ABB RAPID module: ProgSide1.mod

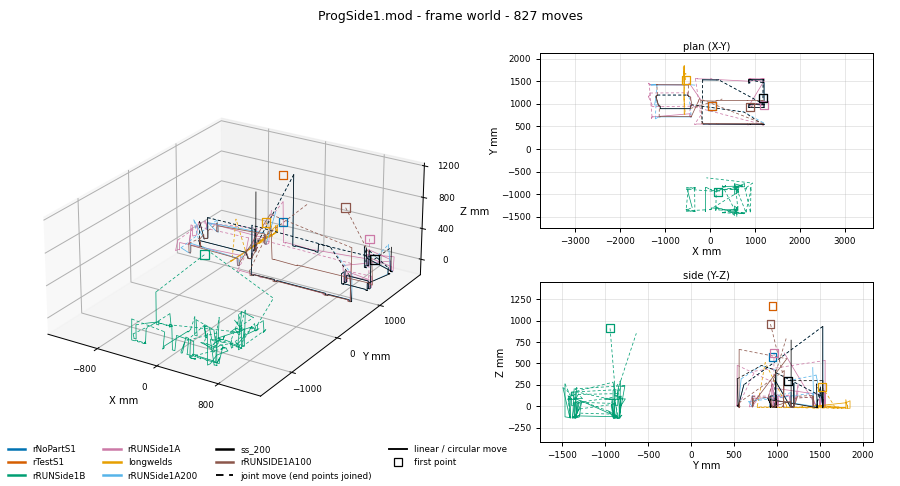
[picture p0: tool path of ProgSide1.mod in frame world, 827 of 843 moves have a stored position in this frame; points joined in program order, loops and branches not executed]
MODULE ProgSide1
    !setup for 300ss
    RECORD WeldPoint300
    robtarget trans;
    robtarget approach;
    robtarget start;
    robtarget end;
    robtarget exitt;
    seamdata seamiii;
    welddata weldiii;
    ENDRECORD
    PERS WeldPoint300 wp300{40};
    PERS num WeldiiiCount := 0;


	!specific zoffset for 200 ss

    TASK PERS wobjdata wobjSide1A200:=[FALSE,TRUE,"",[[0,0,0],[1,0,0,0]],[[0,0,0],[1,0,0,0]]];

    PERS bool bZ_B_onlySide2:=FALSE;
	PERS bool bZ_B_onlySide1:=FALSE;
	PERS bool bC_HalfstepSide2:=FALSE;
	PERS bool bC_HalfstepSide1:=FALSE;
	PERS bool bZ_HalfstepSide1:=FALSE;
	PERS bool bZ_HalfstepSide2:=FALSE;
	PERS bool bAngleSide1:=FALSE;
	PERS bool bAngleSide2:=FALSE;
	PERS bool bTestWeldSide1:=FALSE;
    PERS bool bTestWeldSide2:=FALSE;

    ! Boolian initialization for the SS 300 Frames
    PERS bool bNoPartSide1:=FALSE;
	PERS bool bNoPartSide2:=FALSE;
    PERS bool A_onlySide2:=FALSE;
    PERS bool B_onlySide2:=FALSE;
	PERS bool A_onlySide1:=FALSE;
    PERS bool B_onlySide1:=FALSE;
	PERS bool AB_Side1:=FALSE;
    PERS bool AB_Side2:=FALSE;

    ! Boolian initialization for the SelFrames procedures except the SS 300s.
    PERS bool bSkid50:=FALSE;
    PERS bool bSkid100:=FALSE;
	PERS bool bSkid200:=FALSE;
    PERS bool bSide1A100:=FALSE;
    PERS bool bSide1A200:=FALSE;
    PERS bool bSide1A300:=TRUE;

    PERS bool bRover:=FALSE;
    PERS bool bLongWeld:=FALSE;


	TASK PERS welddata weld7:=[15.24,16.6963,[7,0,0,0,0,0,0,0,0],[7,0,0,0,0,0,0,0,0]];
	TASK PERS welddata weld6:=[16.2983,16.6963,[6,0,0,0,0,0,0,0,0],[6,0,0,0,0,0,0,0,0]];

	CONST robtarget pPounceOS1:=[[-398.58,690.45,580.22],[0.00101632,0.999968,-0.00455572,0.00645523],[-1,0,-1,0],[9E+09,9E+09,9E+09,9E+09,9E+09,9E+09]];
	CONST robtarget pPounceS21:=[[580.19,77.23,83.43],[0.071601,0.767336,-0.436334,0.464416],[-1,0,-2,0],[9E+09,9E+09,9E+09,9E+09,9E+09,9E+09]];
	TASK PERS seamdata seam2:=[4,1,[1,0,52,74.0833,0,0,0,0,0],0,0,0,0,0,[1,0,48,0,0,0,0,0,0],0.01,0.1,[1,0,48,105.833,0,0,0,0,0],0,0,[0,0,0,0,0,0,0,0,0],1];
	TASK PERS seamdata seam10:=[4,1,[1,0,50,80.4333,0,0,0,0,0],0,0,0,0,0,[0,0,0,0,0,0,0,0,0],0.25,0.25,[1,0,50,38.1,0,0,0,0,0],0,0,[0,0,0,0,0,0,0,0,0],1];
	CONST robtarget pPounceS31:=[[358.52,159.10,437.93],[0.0181628,-0.398765,0.916866,0.00362624],[-2,0,-2,0],[9E+09,9E+09,9E+09,9E+09,9E+09,9E+09]];
	CONST robtarget pPounceS41:=[[193.25,136.11,113.74],[0.188325,0.84715,-0.195157,0.45693],[-1,-1,-2,0],[9E+09,9E+09,9E+09,9E+09,9E+09,9E+09]];
	PERS welddata weld11:=[13.5467,0,[1,0,50,84.6667,0,0,0,0,0],[0,0,0,0,0,0,0,0,0]];
	PERS welddata weld10:=[14.8167,0,[1,0,50,95.25,0,0,0,0,0],[0,0,0,0,0,0,0,0,0]];
	TASK PERS seamdata seam11:=[1,1,[1,0,50,84.6667,0,0,0,0,0],0,0,0,0,0,[0,0,0,0,0,0,0,0,0],0,0,[0,0,0,0,0,0,0,0,0],0,0,[0,0,0,0,0,0,0,0,0],0];
	TASK PERS seamdata seam12:=[1,1,[1,0,18.5,381,0,0,0,0,0],0,0,0,0,0,[0,0,0,0,0,0,0,0,0],0,0,[0,0,0,0,0,0,0,0,0],0,0,[0,0,0,0,0,0,0,0,0],0];
	TASK PERS seamdata seam13:=[1,1,[1,0,14,127,0,0,0,0,0],0,0,0,0,0,[0,0,0,0,0,0,0,0,0],0,0,[0,0,0,0,0,0,0,0,0],0,0,[0,0,0,0,0,0,0,0,0],0];
	PERS welddata weld12:=[21.9625,0,[1,0,19,70.6797,0,0,0,0,0],[0,0,0,0,0,0,0,0,0]];
	PERS welddata weld13:=[6.90033,6.90033,[1,0,19,110.71,0,0,0,0,0],[0,0,18.5,110.71,0,0,0,0,0]];
	CONST robtarget pSafeS11:=[[-996.19,963.00,488.78],[0.0459907,-0.688393,0.722625,0.0425673],[1,-1,1,0],[9E+09,9E+09,9E+09,9E+09,9E+09,9E+09]];
	CONST robtarget pSafeS21:=[[-996.19,963.00,488.76],[0.0459983,-0.688397,0.722622,0.0425559],[1,-1,1,0],[9E+09,9E+09,9E+09,9E+09,9E+09,9E+09]];
	CONST robtarget pSafeS31:=[[506.44,675.04,711.34],[0.0314656,-0.935633,0.203865,-0.286426],[0,0,-2,0],[9E+09,9E+09,9E+09,9E+09,9E+09,9E+09]];
	CONST robtarget pSafeS41:=[[488.47,1091.24,654.25],[0.0459806,-0.688392,0.722627,0.0425664],[0,0,-1,0],[9E+09,9E+09,9E+09,9E+09,9E+09,9E+09]];
	CONST robtarget pSafeS51:=[[528.23,1196.89,528.24],[0.224235,-0.753625,-0.525201,-0.325471],[0,-1,-3,0],[9E+09,9E+09,9E+09,9E+09,9E+09,9E+09]];
	CONST robtarget pSafeS61:=[[597.29,1295.03,43.37],[0.191334,-0.732058,-0.538062,-0.371444],[0,-1,-2,0],[9E+09,9E+09,9E+09,9E+09,9E+09,9E+09]];
	CONST robtarget pSafeS71:=[[542.66,1322.39,535.75],[0.223485,-0.764556,-0.487458,-0.357621],[0,-1,-2,0],[9E+09,9E+09,9E+09,9E+09,9E+09,9E+09]];
	CONST robtarget pSafeS81:=[[542.66,1322.38,535.76],[0.223484,-0.764558,-0.487457,-0.35762],[0,-1,-2,0],[9E+09,9E+09,9E+09,9E+09,9E+09,9E+09]];
	CONST robtarget pPounceS51:=[[15.28,993.81,754.75],[0.277209,0.263034,-0.848831,-0.365313],[0,0,0,0],[9E+09,9E+09,9E+09,9E+09,9E+09,9E+09]];
	CONST robtarget pPounceS61:=[[649.55,1131.56,389.19],[0.45355,-0.00505177,-0.879595,-0.143459],[0,0,0,0],[9E+09,9E+09,9E+09,9E+09,9E+09,9E+09]];
	TASK PERS seamdata seam3:=[1,1,[1,0,35,84.6667,0,0,0,0,0],0,0,0,0,0,[1,0,48,0,0,0,0,0,0],0.01,0.1,[1,0,48,105.833,0,0,0,0,0],0,0,[0,0,0,0,0,0,0,0,0],1];
	CONST robtarget pSafeS101:=[[572.94,23.46,738.68],[0.0502756,-0.467207,-0.815726,-0.337314],[0,0,0,0],[9E+09,9E+09,9E+09,9E+09,9E+09,9E+09]];
	CONST robtarget pSafeS111:=[[877.74,-1.14,1156.39],[0.00629855,0.0017594,0.999979,-0.000494623],[0,-1,0,0],[9E+09,9E+09,9E+09,9E+09,9E+09,9E+09]];
	CONST robtarget pSafeS121:=[[877.74,-1.14,1156.39],[0.00629925,0.00175887,0.999979,-0.000492925],[0,-1,0,0],[9E+09,9E+09,9E+09,9E+09,9E+09,9E+09]];
	CONST robtarget pSafeS131:=[[865.02,1139.54,-19.77],[0.144708,-0.274627,0.931028,0.191903],[0,-2,2,0],[9E+09,9E+09,9E+09,9E+09,9E+09,9E+09]];
	CONST robtarget pSafeS141:=[[849.60,1148.97,-24.06],[0.00628216,0.00187497,0.999979,-0.000396021],[0,-1,1,0],[9E+09,9E+09,9E+09,9E+09,9E+09,9E+09]];
	CONST robtarget pSafeS151:=[[1007.97,1505.52,122.27],[0.0460025,-0.688387,0.722632,0.0425454],[0,1,-2,0],[9E+09,9E+09,9E+09,9E+09,9E+09,9E+09]];
	CONST robtarget pHomePos20:=[[365.14,988.92,-33.91],[0.0351389,-0.509982,-0.859022,-0.0276858],[0,-1,1,0],[9E+09,9E+09,9E+09,9E+09,9E+09,9E+09]];
	CONST robtarget pHomePos30:=[[365.15,979.87,-33.91],[0.0351433,-0.509968,-0.85903,-0.0276827],[0,-1,1,0],[9E+09,9E+09,9E+09,9E+09,9E+09,9E+09]];
	CONST robtarget pHomePos40:=[[365.14,979.87,-15.16],[0.0351385,-0.509986,-0.859019,-0.0276867],[0,-1,1,0],[9E+09,9E+09,9E+09,9E+09,9E+09,9E+09]];
	CONST robtarget pHomePos50:=[[433.12,979.73,-15.17],[0.0351369,-0.509964,-0.859032,-0.0276871],[0,-1,1,0],[9E+09,9E+09,9E+09,9E+09,9E+09,9E+09]];
	CONST robtarget pHomePos60:=[[430.57,978.47,-32.25],[0.0351433,-0.50998,-0.859023,-0.0276796],[0,-1,1,0],[9E+09,9E+09,9E+09,9E+09,9E+09,9E+09]];
	CONST robtarget pHomePos70:=[[430.57,978.46,-32.26],[0.0351393,-0.509989,-0.859017,-0.027681],[0,-1,1,0],[9E+09,9E+09,9E+09,9E+09,9E+09,9E+09]];
	CONST robtarget pHomePos80:=[[430.59,974.37,-32.26],[0.0351321,-0.50997,-0.859029,-0.0276862],[0,-1,1,0],[9E+09,9E+09,9E+09,9E+09,9E+09,9E+09]];
	CONST robtarget pHomePos90:=[[430.57,974.36,-24.94],[0.0351397,-0.509992,-0.859016,-0.0276799],[0,-1,1,0],[9E+09,9E+09,9E+09,9E+09,9E+09,9E+09]];
	CONST robtarget pHomePos100:=[[445.83,974.38,-24.94],[0.0351383,-0.509986,-0.859019,-0.0276863],[0,-1,1,0],[9E+09,9E+09,9E+09,9E+09,9E+09,9E+09]];
	CONST robtarget pHomePos110:=[[446.40,974.36,-32.29],[0.0351532,-0.510006,-0.859007,-0.0276708],[0,-1,1,0],[9E+09,9E+09,9E+09,9E+09,9E+09,9E+09]];
	CONST robtarget pHomePos120:=[[446.42,974.37,-32.29],[0.0351424,-0.509994,-0.859014,-0.0276814],[0,-1,1,0],[9E+09,9E+09,9E+09,9E+09,9E+09,9E+09]];
	CONST robtarget pSafeS12:=[[1424.79,-683.57,-13.74],[0.019551,0.168491,0.985501,-0.00412114],[-1,1,-2,0],[9E+09,9E+09,9E+09,9E+09,9E+09,9E+09]];
	CONST robtarget pSafeS22:=[[1462.93,-789.47,-110.40],[0.0637154,0.393325,0.863983,0.307846],[-1,1,-2,0],[9E+09,9E+09,9E+09,9E+09,9E+09,9E+09]];
	CONST robtarget pSafeS32:=[[1462.93,-821.54,-110.39],[0.0637158,0.39332,0.863986,0.307843],[-1,1,-2,0],[9E+09,9E+09,9E+09,9E+09,9E+09,9E+09]];
	CONST robtarget pSafeS42:=[[1462.93,-821.54,-110.39],[0.0637186,0.393326,0.863982,0.307849],[-1,1,-2,0],[9E+09,9E+09,9E+09,9E+09,9E+09,9E+09]];
	CONST robtarget pSafeS52:=[[1462.55,-1477.98,-107.56],[0.0637139,0.393324,0.863983,0.30785],[-1,0,-1,0],[9E+09,9E+09,9E+09,9E+09,9E+09,9E+09]];
	CONST robtarget pSafeS62:=[[1462.54,-1515.56,-107.57],[0.0637098,0.393325,0.863984,0.307846],[-1,0,-1,0],[9E+09,9E+09,9E+09,9E+09,9E+09,9E+09]];
	CONST robtarget pSafeS72:=[[1462.54,-1515.57,-107.57],[0.0637139,0.39333,0.86398,0.307849],[-1,0,-1,0],[9E+09,9E+09,9E+09,9E+09,9E+09,9E+09]];
	CONST robtarget pSafeS82:=[[1462.55,-1515.57,-6.77],[0.063723,0.393334,0.863975,0.307857],[-1,0,-1,0],[9E+09,9E+09,9E+09,9E+09,9E+09,9E+09]];
	CONST robtarget pSafeS161:=[[44.14,948.66,1172.82],[0.0459836,-0.688397,0.722622,0.0425714],[0,-1,0,0],[9E+09,9E+09,9E+09,9E+09,9E+09,9E+09]];
	CONST robtarget pSafeS171:=[[877.68,-1.12,1156.34],[0.00623811,0.00177345,0.999979,-0.000467886],[0,-1,0,0],[9E+09,9E+09,9E+09,9E+09,9E+09,9E+09]];
	CONST robtarget pSafeS181:=[[1178.99,1129.25,299.25],[0.0635535,0.517233,-0.779104,0.348467],[0,1,-3,1],[9E+09,9E+09,9E+09,9E+09,9E+09,9E+09]];
	CONST robtarget pSafeS191:=[[877.68,-1.12,1156.34],[0.00623811,0.00177268,0.999979,-0.000467882],[0,-1,0,0],[9E+09,9E+09,9E+09,9E+09,9E+09,9E+09]];
	CONST robtarget pSafeS201:=[[631.06,-50.80,790.98],[0.377429,-0.0153459,-0.925903,0.00402947],[-1,-1,-5,0],[9E+09,9E+09,9E+09,9E+09,9E+09,9E+09]];
	CONST robtarget pSafeS211:=[[631.06,-50.80,790.98],[0.377429,-0.0153486,-0.925903,0.00403031],[-1,-1,-5,0],[9E+09,9E+09,9E+09,9E+09,9E+09,9E+09]];
	PERS wobjdata wobjShm:=[FALSE,TRUE,"",[[-20,0,0],[1,0,0,0]],[[0,0,0],[1,0,0,0]]];
	CONST robtarget pSafeS221:=[[1178.99,1129.24,299.22],[0.0635644,0.517232,-0.779103,0.348467],[0,1,-2,1],[9E+09,9E+09,9E+09,9E+09,9E+09,9E+09]];
	CONST robtarget pSafeS231:=[[1161.31,998.15,9.10],[0.0635657,0.517232,-0.779104,0.348465],[0,1,-2,1],[9E+09,9E+09,9E+09,9E+09,9E+09,9E+09]];
	CONST robtarget pSafeS241:=[[82.84,919.33,1175.90],[0.326611,0.635475,-0.63738,0.288519],[0,0,-1,0],[9E+09,9E+09,9E+09,9E+09,9E+09,9E+09]];
	CONST robtarget pSafeS251:=[[1164.32,992.14,-2.30],[0.0635629,0.517239,-0.779097,0.348471],[0,1,-2,1],[9E+09,9E+09,9E+09,9E+09,9E+09,9E+09]];
	CONST robtarget pSafeS261:=[[1167.72,990.93,-3.33],[0.0635764,0.517234,-0.779098,0.348472],[0,1,-2,1],[9E+09,9E+09,9E+09,9E+09,9E+09,9E+09]];
	CONST robtarget pSafeS271:=[[1198.72,990.93,-3.32],[0.0635735,0.517235,-0.779098,0.348471],[0,1,-2,1],[9E+09,9E+09,9E+09,9E+09,9E+09,9E+09]];
	CONST robtarget pSafeS281:=[[1004.29,1024.41,280.79],[0.0635732,0.517233,-0.7791,0.34847],[0,1,-2,1],[9E+09,9E+09,9E+09,9E+09,9E+09,9E+09]];


!XXXXXXXXXXXXXXXXXXXXXXXXXXXXXXXXXXXXXXXXXXXXXXXXXXXXXXXXXXXX

!XXXXXXXXXXXXXXXXXXXXXXXXXXXXXXXXXXXXXXXXXXXXXXXXXXXXXXXXXXXX
!xxxxxxxxxxxxxxxxxxxxxxxxxxxxxxxxxxxxxxxxxxxxxxxxxxxxxxxxxxxxxxxx




	PROC rNoPartS1()
		MoveJ pSafeS1, v800, fine, tWeldGun;
		MoveJ pPounceS1, v800, fine, tWeldGun;
		MoveJ pSafeS1, v800, fine, tWeldGun;
	ENDPROC
	PROC rTstA1()
		TPWrite "A S1";
	ENDPROC
	PROC rTstB1()
		TPWrite "B S1";
	ENDPROC
	PROC rTestS1()
		MoveJ [[44.14,948.66,1172.81],[0.0459874,-0.688394,0.722625,0.042569],[0,-1,0,0],[9E+09,9E+09,9E+09,9E+09,9E+09,9E+09]], v1000, z50, tWeldGun;
	ENDPROC
	PROC rRUNSide1B()
		rTestPosTop;
		TPWrite "Side 1 B";
		MoveJ [[173.01,-945.09,908.66],[0.230148,-0.640466,-0.674994,-0.284991],[-1,0,0,0],[9E+09,9E+09,9E+09,9E+09,9E+09,9E+09]], vmax, z50, tWeldGun;
		MoveJ [[-516.56,-891.88,262.76],[0.200577,-0.67934,-0.672798,-0.213563],[-2,0,-1,0],[9E+09,9E+09,9E+09,9E+09,9E+09,9E+09]], vmax, z10, tWeldGun;
		MoveL [[-514.49,-897.92,-127.68],[0.230166,-0.665843,-0.672051,-0.22809],[-2,0,-1,0],[9E+09,9E+09,9E+09,9E+09,9E+09,9E+09]], vmax, z10, tWeldGun;
		ArcLStart [[-513.42,-897.57,-137.38],[0.210753,-0.657323,-0.686354,-0.228973],[-2,0,-1,0],[9E+09,9E+09,9E+09,9E+09,9E+09,9E+09]], v50, seam13, weld13\Weave:=weave1, fine, tWeldGun;
		ArcLEnd [[-481.09,-897.53,-138.19],[0.210743,-0.65735,-0.686326,-0.228987],[-2,0,-1,0],[9E+09,9E+09,9E+09,9E+09,9E+09,9E+09]], v10, seam13, weld13\Weave:=weave1, fine, tWeldGun;
		MoveL [[-479.64,-891.87,-91.90],[0.200495,-0.679391,-0.672743,-0.213649],[-2,0,-1,0],[9E+09,9E+09,9E+09,9E+09,9E+09,9E+09]], vmax, z10, tWeldGun;
		MoveJ [[-526.59,-1340.74,-77.97],[0.272049,0.539222,-0.749573,0.270868],[-2,0,-3,0],[9E+09,9E+09,9E+09,9E+09,9E+09,9E+09]], vmax, z10, tWeldGun;
		MoveL [[-519.95,-1336.21,-124.59],[0.179682,0.6848,-0.680507,0.188877],[-2,-1,-3,0],[9E+09,9E+09,9E+09,9E+09,9E+09,9E+09]], vmax, z10, tWeldGun;
		ArcLStart [[-520.81,-1338.24,-133.17],[0.193377,0.681101,-0.684106,0.175232],[-2,-1,-3,0],[9E+09,9E+09,9E+09,9E+09,9E+09,9E+09]], v50, seam13, weld13\Weave:=weave1, fine, tWeldGun;
		ArcLEnd [[-489.52,-1337.73,-131.66],[0.193296,0.681188,-0.684044,0.175225],[-2,-1,-3,0],[9E+09,9E+09,9E+09,9E+09,9E+09,9E+09]], v10, seam13, weld13\Weave:=weave1, fine, tWeldGun;
		MoveL [[-484.84,-1342.71,46.50],[0.235633,0.655478,-0.679432,0.230648],[-2,-1,-3,0],[9E+09,9E+09,9E+09,9E+09,9E+09,9E+09]], vmax, z10, tWeldGun;
		MoveJ [[-392.56,-1296.67,69.52],[0.264192,0.731229,-0.303703,0.550702],[-2,0,0,0],[9E+09,9E+09,9E+09,9E+09,9E+09,9E+09]], vmax, z20, tWeldGun;
		MoveL [[-512.18,-856.47,-124.70],[0.238884,-0.653044,-0.673688,-0.250226],[-2,0,-1,0],[9E+09,9E+09,9E+09,9E+09,9E+09,9E+09]], vmax, z10, tWeldGun;
		ArcLStart [[-513.54,-858.91,-136.72],[0.215398,-0.662814,-0.680722,-0.225612],[-2,0,-1,0],[9E+09,9E+09,9E+09,9E+09,9E+09,9E+09]], v50, seam13, weld13, fine, tWeldGun;
		ArcLEnd [[-473.42,-859.48,-137.35],[0.215439,-0.662758,-0.68077,-0.22559],[-2,0,-1,0],[9E+09,9E+09,9E+09,9E+09,9E+09,9E+09]], v10, seam13, weld13\Weave:=weave1, fine, tWeldGun;
		MoveL [[-470.56,-868.46,-128.98],[0.215449,-0.66272,-0.680808,-0.225579],[-2,0,-1,0],[9E+09,9E+09,9E+09,9E+09,9E+09,9E+09]], vmax, z10, tWeldGun;
		MoveL [[-436.87,-865.82,-129.01],[0.215414,-0.662677,-0.680771,-0.225849],[-2,0,-1,0],[9E+09,9E+09,9E+09,9E+09,9E+09,9E+09]], vmax, z10, tWeldGun;
		ArcLStart [[-436.92,-859.84,-136.80],[0.215444,-0.662646,-0.680803,-0.225813],[-2,0,-1,0],[9E+09,9E+09,9E+09,9E+09,9E+09,9E+09]], v50, seam13, weld13\Weave:=weave1, fine, tWeldGun;
		ArcLEnd [[-395.30,-860.19,-135.58],[0.21546,-0.662716,-0.680804,-0.225593],[-2,0,-1,0],[9E+09,9E+09,9E+09,9E+09,9E+09,9E+09]], v10, seam13, weld13\Weave:=weave1, fine, tWeldGun;
		MoveL [[-394.28,-872.79,-127.38],[0.215463,-0.66272,-0.6808,-0.225589],[-2,0,-1,0],[9E+09,9E+09,9E+09,9E+09,9E+09,9E+09]], vmax, z10, tWeldGun;
		MoveL [[-366.90,-866.62,-125.77],[0.215457,-0.662713,-0.680808,-0.225591],[-2,0,-1,0],[9E+09,9E+09,9E+09,9E+09,9E+09,9E+09]], vmax, z10, tWeldGun;
		ArcLStart [[-366.93,-860.65,-137.16],[0.215461,-0.662729,-0.680792,-0.225588],[-2,0,-1,0],[9E+09,9E+09,9E+09,9E+09,9E+09,9E+09]], v50, seam13, weld13\Weave:=weave1, fine, tWeldGun;
		ArcLEnd [[-338.32,-860.21,-136.79],[0.215451,-0.662739,-0.68078,-0.225604],[-2,0,-1,0],[9E+09,9E+09,9E+09,9E+09,9E+09,9E+09]], v10, seam13, weld13\Weave:=weave1, fine, tWeldGun;
		MoveL [[-339.56,-873.86,-125.98],[0.215452,-0.662777,-0.680806,-0.225413],[-2,0,-1,0],[9E+09,9E+09,9E+09,9E+09,9E+09,9E+09]], vmax, z10, tWeldGun;
		MoveL [[-336.25,-871.19,-128.23],[0.0916487,-0.841258,-0.420907,-0.326687],[-2,0,-1,0],[9E+09,9E+09,9E+09,9E+09,9E+09,9E+09]], vmax, z10, tWeldGun;
		ArcLStart [[-335.10,-862.58,-134.24],[0.0916576,-0.841254,-0.420918,-0.326679],[-2,0,-1,0],[9E+09,9E+09,9E+09,9E+09,9E+09,9E+09]], v50, seam13, weld13, fine, tWeldGun;
		ArcLEnd [[-339.89,-887.39,-134.70],[0.00906284,0.920107,0.0370263,0.389808],[-2,0,0,0],[9E+09,9E+09,9E+09,9E+09,9E+09,9E+09]], v10, seam13, weld13, fine, tWeldGun;
		MoveL [[-340.52,-888.78,-94.76],[0.0606807,0.91536,0.0671192,0.392339],[-2,0,0,0],[9E+09,9E+09,9E+09,9E+09,9E+09,9E+09]], v100, z10, tWeldGun;
		MoveL [[-322.29,-862.50,-115.71],[0.124255,-0.837706,-0.434858,-0.306118],[-2,0,0,0],[9E+09,9E+09,9E+09,9E+09,9E+09,9E+09]], v100, z10, tWeldGun;
		ArcLStart [[-317.89,-862.07,-130.90],[0.120916,-0.838204,-0.433585,-0.307894],[-2,0,0,0],[9E+09,9E+09,9E+09,9E+09,9E+09,9E+09]], v10, seam13, weld13\Weave:=weave1, fine, tWeldGun;
		ArcLEnd [[-337.44,-859.45,-134.89],[0.12429,-0.837713,-0.434783,-0.306193],[-2,0,0,0],[9E+09,9E+09,9E+09,9E+09,9E+09,9E+09]], v10, seam13, weld13\Weave:=weave1, fine, tWeldGun;
		MoveL [[-337.89,-880.77,33.09],[0.124309,-0.837706,-0.434822,-0.306146],[-2,0,0,0],[9E+09,9E+09,9E+09,9E+09,9E+09,9E+09]], vmax, z10, tWeldGun;
		MoveJ [[-332.34,-1363.85,48.88],[0.219066,0.836756,-0.390875,0.31475],[-2,-1,1,0],[9E+09,9E+09,9E+09,9E+09,9E+09,9E+09]], vmax, z10, tWeldGun;
		MoveL [[-348.32,-1358.04,-125.11],[0.0288552,0.954843,-0.0190534,0.295092],[-2,-1,1,0],[9E+09,9E+09,9E+09,9E+09,9E+09,9E+09]], vmax, z10, tWeldGun;
		ArcLStart [[-347.38,-1361.16,-134.40],[0.0287871,0.954854,-0.0190038,0.295067],[-2,-1,1,0],[9E+09,9E+09,9E+09,9E+09,9E+09,9E+09]], v50, seam13, weld13\Weave:=weave1, fine, tWeldGun;
		ArcLEnd [[-347.45,-1384.56,-132.93],[0.145016,0.917129,-0.235371,0.287135],[-2,-1,1,0],[9E+09,9E+09,9E+09,9E+09,9E+09,9E+09]], v10, seam13, weld13\Weave:=weave1, fine, tWeldGun;
		MoveL [[-345.43,-1382.83,-124.95],[0.145024,0.917114,-0.235421,0.287137],[-2,-1,1,0],[9E+09,9E+09,9E+09,9E+09,9E+09,9E+09]], vmax, z10, tWeldGun;
		MoveL [[-328.65,-1384.41,-121.55],[0.145003,0.917127,-0.235391,0.287129],[-2,-1,1,0],[9E+09,9E+09,9E+09,9E+09,9E+09,9E+09]], vmax, z10, tWeldGun;
		ArcLStart [[-324.47,-1384.79,-126.79],[0.144984,0.917133,-0.235388,0.287122],[-2,-1,1,0],[9E+09,9E+09,9E+09,9E+09,9E+09,9E+09]], v10, seam13, weld13\Weave:=weave1, fine, tWeldGun;
		ArcLEnd [[-349.04,-1384.95,-130.97],[0.144974,0.917151,-0.235337,0.287113],[-2,-1,1,0],[9E+09,9E+09,9E+09,9E+09,9E+09,9E+09]], v10, seam13, weld13\Weave:=weave1, fine, tWeldGun;
		MoveL [[-350.83,-1367.95,-122.57],[0.144998,0.917131,-0.235387,0.287125],[-2,-1,1,0],[9E+09,9E+09,9E+09,9E+09,9E+09,9E+09]], vmax, z10, tWeldGun;
		MoveL [[-341.99,-1371.18,-117.57],[0.232266,0.668561,-0.669899,0.224308],[-2,-1,1,0],[9E+09,9E+09,9E+09,9E+09,9E+09,9E+09]], vmax, z10, tWeldGun;
		ArcLStart [[-346.33,-1380.76,-134.98],[0.232264,0.668628,-0.669837,0.224295],[-2,-1,1,0],[9E+09,9E+09,9E+09,9E+09,9E+09,9E+09]], v30, seam13, weld13, fine, tWeldGun;
		ArcLEnd [[-381.42,-1380.97,-134.58],[0.232255,0.668596,-0.66987,0.224303],[-2,-1,1,0],[9E+09,9E+09,9E+09,9E+09,9E+09,9E+09]], v10, seam13, weld13, fine, tWeldGun;
		MoveL [[-381.43,-1374.36,-128.77],[0.232262,0.668602,-0.669863,0.224299],[-2,-1,1,0],[9E+09,9E+09,9E+09,9E+09,9E+09,9E+09]], vmax, z10, tWeldGun;
		MoveL [[-417.42,-1374.56,-128.76],[0.232259,0.668611,-0.669855,0.224298],[-2,-1,1,0],[9E+09,9E+09,9E+09,9E+09,9E+09,9E+09]], vmax, z10, tWeldGun;
		ArcLStart [[-417.87,-1380.73,-134.98],[0.232273,0.668637,-0.669829,0.224284],[-2,-1,1,0],[9E+09,9E+09,9E+09,9E+09,9E+09,9E+09]], v50, seam13, weld13\Weave:=weave1, fine, tWeldGun;
		ArcLEnd [[-444.46,-1379.77,-134.96],[0.232272,0.668636,-0.669829,0.224287],[-2,-1,1,0],[9E+09,9E+09,9E+09,9E+09,9E+09,9E+09]], v10, seam13, weld13\Weave:=weave1, fine, tWeldGun;
		MoveL [[-444.47,-1371.57,-127.54],[0.232274,0.66863,-0.669834,0.224288],[-2,-1,1,0],[9E+09,9E+09,9E+09,9E+09,9E+09,9E+09]], vmax, z10, tWeldGun;
		MoveL [[-474.23,-1371.36,-127.53],[0.232273,0.668635,-0.66983,0.224288],[-2,-1,1,0],[9E+09,9E+09,9E+09,9E+09,9E+09,9E+09]], vmax, z10, tWeldGun;
		ArcLStart [[-474.48,-1379.73,-134.16],[0.232266,0.668654,-0.669817,0.224275],[-2,-1,1,0],[9E+09,9E+09,9E+09,9E+09,9E+09,9E+09]], v50, seam13, weld13\Weave:=weave1, fine, tWeldGun;
		ArcLEnd [[-520.49,-1380.65,-135.20],[0.232213,0.668741,-0.669751,0.224268],[-2,-1,1,0],[9E+09,9E+09,9E+09,9E+09,9E+09,9E+09]], v10, seam13, weld13\Weave:=weave1, fine, tWeldGun;
		MoveL [[-521.34,-1368.99,120.05],[0.232497,0.668664,-0.669682,0.22441],[-2,-1,1,0],[9E+09,9E+09,9E+09,9E+09,9E+09,9E+09]], vmax, z10, tWeldGun;
		MoveJ [[-94.49,-1349.72,64.27],[0.311518,0.0288903,-0.949685,-0.0148846],[-2,0,-2,0],[9E+09,9E+09,9E+09,9E+09,9E+09,9E+09]], vmax, z10, tWeldGun;
		MoveL [[-94.58,-1386.97,-127.39],[0.311577,0.0288594,-0.949671,-0.0145439],[-2,0,-2,0],[9E+09,9E+09,9E+09,9E+09,9E+09,9E+09]], vmax, z10, tWeldGun;
		ArcLStart [[-100.40,-1387.16,-133.37],[0.311603,0.0288403,-0.949663,-0.0145528],[-2,0,-2,0],[9E+09,9E+09,9E+09,9E+09,9E+09,9E+09]], v50, seam13, weld13\Weave:=weave1, fine, tWeldGun;
		ArcLEnd [[-99.80,-1356.97,-133.39],[0.311608,0.0288143,-0.949662,-0.0145611],[-2,0,-2,0],[9E+09,9E+09,9E+09,9E+09,9E+09,9E+09]], v10, seam13, weld13\Weave:=weave1, fine, tWeldGun;
		MoveL [[-99.63,-1357.12,-110.82],[0.311637,0.0288227,-0.949655,-0.014427],[-2,0,-2,0],[9E+09,9E+09,9E+09,9E+09,9E+09,9E+09]], vmax, z10, tWeldGun;
		!MoveJ [[-89.18,-890.48,-106.53],[0.311095,0.0172745,-0.950222,-0.000691898],[-2,0,-2,0],[9E+09,9E+09,9E+09,9E+09,9E+09,9E+09]], vmax, z10, tWeldGun;
		MoveL [[-92.20,-882.67,-120.77],[0.311167,0.0172923,-0.950198,-0.000589398],[-2,0,-2,0],[9E+09,9E+09,9E+09,9E+09,9E+09,9E+09]], vmax, z10, tWeldGun;
		ArcLStart [[-97.41,-881.04,-134.98],[0.311176,0.0172867,-0.950195,-0.000618972],[-2,0,-2,0],[9E+09,9E+09,9E+09,9E+09,9E+09,9E+09]], v50, seam13, weld13\Weave:=weave1, fine, tWeldGun;
		ArcLEnd [[-97.13,-850.24,-135.19],[0.31116,0.0171976,-0.950202,-0.000643122],[-2,0,-2,0],[9E+09,9E+09,9E+09,9E+09,9E+09,9E+09]], v10, seam13, weld13\Weave:=weave1, fine, tWeldGun;
		MoveL [[-76.90,-853.66,-105.59],[0.311086,0.0173184,-0.950224,-0.000798945],[-2,0,-2,0],[9E+09,9E+09,9E+09,9E+09,9E+09,9E+09]], vmax, z10, tWeldGun;
		MoveJ [[5.08,-892.16,87.65],[0.246917,-0.649526,-0.670091,-0.261011],[-2,0,-1,0],[9E+09,9E+09,9E+09,9E+09,9E+09,9E+09]], vmax, z10, tWeldGun;
		MoveL [[5.70,-898.13,-125.58],[0.246931,-0.64953,-0.670081,-0.261012],[-2,0,-1,0],[9E+09,9E+09,9E+09,9E+09,9E+09,9E+09]], vmax, z10, tWeldGun;
		ArcLStart [[5.31,-898.71,-138.77],[0.203028,-0.669224,-0.681322,-0.21615],[-2,0,-1,0],[9E+09,9E+09,9E+09,9E+09,9E+09,9E+09]], v50, seam13, weld13\Weave:=weave1, fine, tWeldGun;
		ArcLEnd [[39.10,-899.19,-140.54],[0.203016,-0.669237,-0.681312,-0.216149],[-1,0,-1,0],[9E+09,9E+09,9E+09,9E+09,9E+09,9E+09]], v10, seam13, weld13\Weave:=weave1, fine, tWeldGun;
		MoveL [[40.66,-920.62,70.48],[0.246699,-0.649617,-0.670207,-0.260692],[-1,0,-1,0],[9E+09,9E+09,9E+09,9E+09,9E+09,9E+09]], vmax, z10, tWeldGun;
		MoveJ [[283.83,-931.65,13.13],[0.246958,-0.649486,-0.670134,-0.26096],[-1,0,0,0],[9E+09,9E+09,9E+09,9E+09,9E+09,9E+09]], vmax, z10, tWeldGun;
		MoveL [[286.40,-910.85,-115.99],[0.24696,-0.649475,-0.670149,-0.260949],[-1,0,0,0],[9E+09,9E+09,9E+09,9E+09,9E+09,9E+09]], vmax, z10, tWeldGun;
		ArcLStart [[286.60,-900.05,-139.30],[0.199989,-0.665549,-0.686307,-0.214554],[-1,-1,0,0],[9E+09,9E+09,9E+09,9E+09,9E+09,9E+09]], v50, seam13, weld13\Weave:=weave1, fine, tWeldGun;
		ArcLEnd [[317.15,-902.62,-138.51],[0.20006,-0.6655,-0.686344,-0.21452],[-1,-1,0,0],[9E+09,9E+09,9E+09,9E+09,9E+09,9E+09]], v10, seam13, weld13\Weave:=weave1, fine, tWeldGun;
		MoveL [[324.35,-903.06,-116.80],[0.246972,-0.649396,-0.670267,-0.260831],[-1,0,0,0],[9E+09,9E+09,9E+09,9E+09,9E+09,9E+09]], vmax, z10, tWeldGun;
		MoveJ [[559.57,-898.83,-116.82],[0.246966,-0.649476,-0.670148,-0.260944],[-1,-1,0,0],[9E+09,9E+09,9E+09,9E+09,9E+09,9E+09]], vmax, z10, tWeldGun;
		MoveL [[560.55,-906.62,-132.43],[0.246958,-0.649466,-0.670157,-0.260952],[-1,-1,0,0],[9E+09,9E+09,9E+09,9E+09,9E+09,9E+09]], vmax, z10, tWeldGun;
		ArcLStart [[565.11,-902.42,-135.83],[0.247002,-0.649431,-0.670186,-0.260923],[-1,-1,0,0],[9E+09,9E+09,9E+09,9E+09,9E+09,9E+09]], v50, seam13, weld13\Weave:=weave1, fine, tWeldGun;
		ArcLEnd [[597.09,-902.15,-136.44],[0.247046,-0.649416,-0.670188,-0.260912],[-1,-1,0,0],[9E+09,9E+09,9E+09,9E+09,9E+09,9E+09]], v10, seam13, weld13\Weave:=weave1, fine, tWeldGun;
		MoveL [[596.75,-960.43,-56.34],[0.246991,-0.649449,-0.670174,-0.260919],[-1,-1,0,0],[9E+09,9E+09,9E+09,9E+09,9E+09,9E+09]], vmax, z10, tWeldGun;
		MoveJ [[601.82,-903.83,-123.32],[0.326164,-0.613251,-0.630337,-0.346722],[-1,0,0,0],[9E+09,9E+09,9E+09,9E+09,9E+09,9E+09]], vmax, z10, tWeldGun;
		MoveL [[600.91,-903.21,-128.01],[0.274675,-0.639039,-0.654325,-0.296719],[-1,0,0,0],[9E+09,9E+09,9E+09,9E+09,9E+09,9E+09]], v100, z10, tWeldGun;
		ArcLStart [[599.42,-898.47,-136.03],[0.274711,-0.63902,-0.654345,-0.296683],[-1,0,0,0],[9E+09,9E+09,9E+09,9E+09,9E+09,9E+09]], v10, seam13, weld13\Weave:=weave1, fine, tWeldGun;
		ArcLEnd [[632.42,-900.13,-136.04],[0.274755,-0.638991,-0.654368,-0.296653],[-1,0,0,0],[9E+09,9E+09,9E+09,9E+09,9E+09,9E+09]], v10, seam13, weld13\Weave:=weave1, fine, tWeldGun;
		MoveL [[633.74,-910.04,-132.93],[0.326202,-0.613258,-0.630325,-0.346695],[-1,0,0,0],[9E+09,9E+09,9E+09,9E+09,9E+09,9E+09]], vmax, z10, tWeldGun;
		MoveL [[633.73,-910.04,183.03],[0.326216,-0.613247,-0.630334,-0.346685],[-1,0,0,0],[9E+09,9E+09,9E+09,9E+09,9E+09,9E+09]], vmax, z10, tWeldGun;
		MoveJ [[627.00,-822.44,298.30],[0.361159,0.600904,-0.609737,0.36973],[-1,-1,-2,0],[9E+09,9E+09,9E+09,9E+09,9E+09,9E+09]], vmax, z10, tWeldGun;
		MoveL [[624.89,-836.84,-138.33],[0.402446,0.574392,-0.586393,0.405284],[-1,-2,-1,0],[9E+09,9E+09,9E+09,9E+09,9E+09,9E+09]], vmax, z10, tWeldGun;
		ArcLStart [[629.25,-851.26,-137.07],[0.402491,0.574255,-0.586521,0.405249],[-1,-2,-1,0],[9E+09,9E+09,9E+09,9E+09,9E+09,9E+09]], v50, seam13, weld13\Weave:=weave1, fine, tWeldGun;
		ArcLEnd [[596.80,-848.27,-137.48],[0.4025,0.574227,-0.586557,0.405227],[-1,-2,-1,0],[9E+09,9E+09,9E+09,9E+09,9E+09,9E+09]], v10, seam13, weld13\Weave:=weave1, fine, tWeldGun;
		MoveL [[595.98,-827.09,-135.34],[0.402393,0.574513,-0.586267,0.405347],[-1,-2,-1,0],[9E+09,9E+09,9E+09,9E+09,9E+09,9E+09]], vmax, z10, tWeldGun;
		MoveL [[627.09,-846.85,78.98],[0.483059,0.507565,-0.528798,0.478963],[-1,-2,-1,0],[9E+09,9E+09,9E+09,9E+09,9E+09,9E+09]], vmax, z10, tWeldGun;
		ArcLStart [[626.96,-857.86,79.00],[0.483055,0.507564,-0.52879,0.478977],[-1,-2,-1,0],[9E+09,9E+09,9E+09,9E+09,9E+09,9E+09]], v40, seam13, weld13\Weave:=weave1, fine, tWeldGun;
		ArcLEnd [[593.04,-858.07,78.79],[0.483033,0.507633,-0.52873,0.478992],[-1,-2,-1,0],[9E+09,9E+09,9E+09,9E+09,9E+09,9E+09]], v10, seam13, weld13\Weave:=weave1, fine, tWeldGun;
		MoveL [[594.80,-840.42,83.53],[0.487698,0.503251,-0.532984,0.47415],[-1,-2,-1,0],[9E+09,9E+09,9E+09,9E+09,9E+09,9E+09]], vmax, z10, tWeldGun;
		SingArea\Wrist;
		MoveJ [[510.38,-859.01,160.69],[0.00485322,0.746032,-0.024255,0.665452],[-1,0,0,0],[9E+09,9E+09,9E+09,9E+09,9E+09,9E+09]], vmax, z10, tWeldGun;
		MoveL [[590.96,-857.11,78.44],[0.00482135,0.745929,-0.024224,0.665567],[-1,0,0,0],[9E+09,9E+09,9E+09,9E+09,9E+09,9E+09]], vmax, z10, tWeldGun;
		ArcLStart [[598.52,-857.62,79.43],[0.0048762,0.74592,-0.0242869,0.665576],[-1,0,0,0],[9E+09,9E+09,9E+09,9E+09,9E+09,9E+09]], v40, seam13, weld13\Weave:=weave1, fine, tWeldGun;
		ArcLEnd [[598.28,-891.23,79.40],[0.00487751,0.745929,-0.0242988,0.665564],[-1,0,0,0],[9E+09,9E+09,9E+09,9E+09,9E+09,9E+09]], v10, seam13, weld13\Weave:=weave1, fine, tWeldGun;
		MoveL [[545.64,-889.59,83.73],[0.0047987,0.745982,-0.0242261,0.665508],[-1,0,0,0],[9E+09,9E+09,9E+09,9E+09,9E+09,9E+09]], vmax, z10, tWeldGun;
		MoveL [[545.47,-1007.73,83.69],[0.00477345,0.745999,-0.0242032,0.665491],[-1,0,0,0],[9E+09,9E+09,9E+09,9E+09,9E+09,9E+09]], vmax, z10, tWeldGun;
		MoveJ [[631.13,-962.99,83.64],[0.467638,-0.538268,-0.512971,-0.477958],[-1,0,0,0],[9E+09,9E+09,9E+09,9E+09,9E+09,9E+09]], vmax, z10, tWeldGun;
		MoveL [[598.78,-893.01,80.08],[0.467241,-0.531733,-0.519718,-0.478373],[-1,0,0,0],[9E+09,9E+09,9E+09,9E+09,9E+09,9E+09]], vmax, z10, tWeldGun;
		ArcLStart [[597.58,-887.83,80.09],[0.467245,-0.531734,-0.519718,-0.478366],[-1,0,0,0],[9E+09,9E+09,9E+09,9E+09,9E+09,9E+09]], v50, seam13, weld13\Weave:=weave1, fine, tWeldGun;
		ArcLEnd [[631.17,-888.01,80.07],[0.467243,-0.531739,-0.519697,-0.478386],[-1,0,0,0],[9E+09,9E+09,9E+09,9E+09,9E+09,9E+09]], v10, seam13, weld13\Weave:=weave1, fine, tWeldGun;
		MoveL [[633.84,-953.29,84.81],[0.467086,-0.531839,-0.51974,-0.478381],[-1,0,0,0],[9E+09,9E+09,9E+09,9E+09,9E+09,9E+09]], vmax, z10, tWeldGun;
		MoveJ [[-0.34,-1346.80,171.20],[0.287604,0.644423,-0.651566,0.278325],[-1,-1,-2,0],[9E+09,9E+09,9E+09,9E+09,9E+09,9E+09]], vmax, z10, tWeldGun;
		MoveL [[-2.14,-1338.76,-121.61],[0.287464,0.644565,-0.651541,0.278198],[-1,-1,-2,0],[9E+09,9E+09,9E+09,9E+09,9E+09,9E+09]], vmax, z10, tWeldGun;
		ArcLStart [[-0.76,-1343.80,-136.83],[0.245347,0.661449,-0.666192,0.241824],[-1,0,-2,0],[9E+09,9E+09,9E+09,9E+09,9E+09,9E+09]], v40, seam13, weld13\Weave:=weave1, fine, tWeldGun;
		ArcLEnd [[33.80,-1343.62,-136.84],[0.226607,0.667964,-0.672794,0.223208],[-1,0,-2,0],[9E+09,9E+09,9E+09,9E+09,9E+09,9E+09]], v10, seam13, weld13\Weave:=weave1, fine, tWeldGun;
		MoveL [[33.45,-1306.76,35.10],[0.287609,0.644475,-0.651512,0.278328],[-1,-1,-2,0],[9E+09,9E+09,9E+09,9E+09,9E+09,9E+09]], vmax, z10, tWeldGun;
		MoveL [[273.41,-1327.02,35.12],[0.287608,0.6445,-0.651487,0.278327],[-1,-1,-2,0],[9E+09,9E+09,9E+09,9E+09,9E+09,9E+09]], vmax, z10, tWeldGun;
		MoveL [[281.49,-1342.97,-129.04],[0.226085,0.668734,-0.671173,0.226292],[-1,0,-2,0],[9E+09,9E+09,9E+09,9E+09,9E+09,9E+09]], vmax, z10, tWeldGun;
		ArcLStart [[279.71,-1344.95,-134.87],[0.226101,0.66872,-0.671191,0.226263],[-1,0,-2,0],[9E+09,9E+09,9E+09,9E+09,9E+09,9E+09]], v40, seam13, weld13\Weave:=weave1, fine, tWeldGun;
		ArcLEnd [[313.39,-1345.44,-135.63],[0.216572,0.670482,-0.675602,0.217056],[-1,0,-2,0],[9E+09,9E+09,9E+09,9E+09,9E+09,9E+09]], v10, seam13, weld13\Weave:=weave1, fine, tWeldGun;
		MoveL [[313.56,-1350.36,-117.72],[0.287596,0.644518,-0.651477,0.278324],[-1,-1,-2,0],[9E+09,9E+09,9E+09,9E+09,9E+09,9E+09]], vmax, z10, tWeldGun;
		MoveL [[559.03,-1342.37,-128.81],[0.261338,0.655204,-0.662463,0.2521],[-1,0,-2,0],[9E+09,9E+09,9E+09,9E+09,9E+09,9E+09]], vmax, z10, tWeldGun;
		ArcLStart [[559.28,-1346.89,-135.25],[0.237304,0.663875,-0.671451,0.228278],[-1,0,-2,0],[9E+09,9E+09,9E+09,9E+09,9E+09,9E+09]], v40, seam13, weld13\Weave:=weave1, fine, tWeldGun;
		ArcLEnd [[593.61,-1347.58,-135.07],[0.242706,0.662076,-0.669468,0.233586],[-1,0,-2,0],[9E+09,9E+09,9E+09,9E+09,9E+09,9E+09]], v10, seam13, weld13\Weave:=weave1, fine, tWeldGun;
		MoveL [[591.10,-1294.92,-96.48],[0.287644,0.644544,-0.6514,0.278391],[-1,-1,-2,0],[9E+09,9E+09,9E+09,9E+09,9E+09,9E+09]], vmax, z10, tWeldGun;
		!MoveJ [[629.17,-1265.05,-98.00],[0.340013,0.628245,-0.617658,0.328935],[-1,-1,-2,0],[9E+09,9E+09,9E+09,9E+09,9E+09,9E+09]], vmax, z10, tWeldGun;
		MoveL [[591.41,-1351.39,-134.59],[0.327693,0.635442,-0.623094,0.31715],[-1,-1,-2,0],[9E+09,9E+09,9E+09,9E+09,9E+09,9E+09]], vmax, z10, tWeldGun;
		ArcLStart [[593.62,-1352.37,-134.75],[0.327705,0.635467,-0.623058,0.31716],[-1,-1,-2,0],[9E+09,9E+09,9E+09,9E+09,9E+09,9E+09]], v40, seam13, weld13\Weave:=weave1, fine, tWeldGun;
		ArcLEnd [[621.10,-1352.20,-134.97],[0.327706,0.635474,-0.623058,0.317146],[-1,-1,-2,0],[9E+09,9E+09,9E+09,9E+09,9E+09,9E+09]], v10, seam13, weld13\Weave:=weave1, fine, tWeldGun;
		MoveL [[594.26,-1304.04,-124.90],[0.375061,0.603881,-0.605571,0.35769],[-1,-1,-2,0],[9E+09,9E+09,9E+09,9E+09,9E+09,9E+09]], vmax, z10, tWeldGun;
		MoveL [[623.93,-1279.28,49.33],[0.327728,0.635484,-0.623033,0.31715],[-1,-1,-2,0],[9E+09,9E+09,9E+09,9E+09,9E+09,9E+09]], vmax, z10, tWeldGun;
		MoveJ [[598.90,-1494.47,216.89],[0.17643,-0.701594,-0.668329,-0.173135],[-1,-1,0,0],[9E+09,9E+09,9E+09,9E+09,9E+09,9E+09]], vmax, z10, tWeldGun;
		MoveL [[594.87,-1413.54,-135.44],[0.380481,-0.610449,-0.582556,-0.378439],[-1,0,0,0],[9E+09,9E+09,9E+09,9E+09,9E+09,9E+09]], vmax, z10, tWeldGun;
		ArcLStart [[597.44,-1406.59,-134.67],[0.380391,-0.610521,-0.582612,-0.378326],[-1,0,0,0],[9E+09,9E+09,9E+09,9E+09,9E+09,9E+09]], v50, seam13, weld13\Weave:=weave1, fine, tWeldGun;
		ArcLEnd [[626.78,-1404.58,-135.67],[0.380425,-0.610529,-0.582583,-0.378324],[-1,0,0,0],[9E+09,9E+09,9E+09,9E+09,9E+09,9E+09]], v10, seam13, weld13\Weave:=weave1, fine, tWeldGun;
		MoveL [[628.35,-1412.36,-131.21],[0.467542,-0.524114,-0.539124,-0.464817],[-1,0,0,0],[9E+09,9E+09,9E+09,9E+09,9E+09,9E+09]], vmax, z10, tWeldGun;
		MoveL [[630.04,-1413.39,82.24],[0.406954,-0.557371,-0.567573,-0.448985],[-1,0,0,0],[9E+09,9E+09,9E+09,9E+09,9E+09,9E+09]], vmax, z10, tWeldGun;
		ArcLStart [[628.70,-1401.58,82.12],[0.406984,-0.557334,-0.567484,-0.449117],[-1,0,0,0],[9E+09,9E+09,9E+09,9E+09,9E+09,9E+09]], v40, seam13, weld13\Weave:=weave1, fine, tWeldGun;
		ArcLEnd [[596.09,-1401.19,82.09],[0.406987,-0.557342,-0.567472,-0.44912],[-1,0,0,0],[9E+09,9E+09,9E+09,9E+09,9E+09,9E+09]], v10, seam13, weld13\Weave:=weave1, fine, tWeldGun;
		MoveL [[597.75,-1438.39,81.60],[0.377561,-0.521089,-0.645673,-0.411121],[-1,0,0,0],[9E+09,9E+09,9E+09,9E+09,9E+09,9E+09]], vmax, z10, tWeldGun;
		MoveL [[409.08,-1390.23,81.60],[0.377566,-0.521097,-0.645665,-0.411119],[-1,0,0,0],[9E+09,9E+09,9E+09,9E+09,9E+09,9E+09]], vmax, z10, tWeldGun;
		MoveJ [[483.55,-1400.78,96.25],[0.150969,0.719954,0.110873,0.668268],[-1,0,0,0],[9E+09,9E+09,9E+09,9E+09,9E+09,9E+09]], vmax, z10, tWeldGun;
		MoveL [[586.16,-1400.86,80.98],[0.0313045,0.743014,0.0228137,0.668155],[-1,0,0,0],[9E+09,9E+09,9E+09,9E+09,9E+09,9E+09]], vmax, z10, tWeldGun;
		ArcLStart [[591.64,-1402.95,82.31],[0.0312871,0.743046,0.0227572,0.668122],[-1,0,0,0],[9E+09,9E+09,9E+09,9E+09,9E+09,9E+09]], v50, seam13, weld13\Weave:=weave1, fine, tWeldGun;
		ArcLEnd [[593.22,-1369.37,81.89],[0.0312913,0.74305,0.0227464,0.668117],[-1,0,0,0],[9E+09,9E+09,9E+09,9E+09,9E+09,9E+09]], v10, seam13, weld13\Weave:=weave1, fine, tWeldGun;
		MoveL [[554.18,-1372.28,89.73],[0.15109,0.720146,0.110407,0.668112],[-1,0,0,0],[9E+09,9E+09,9E+09,9E+09,9E+09,9E+09]], vmax, z10, tWeldGun;
		MoveL [[549.71,-1268.25,89.71],[0.151117,0.720151,0.110329,0.668113],[-1,1,0,0],[9E+09,9E+09,9E+09,9E+09,9E+09,9E+09]], vmax, z10, tWeldGun;
		MoveJ [[603.39,-1313.43,143.58],[0.469159,0.533622,-0.523436,0.470269],[-1,-2,3,0],[9E+09,9E+09,9E+09,9E+09,9E+09,9E+09]], vmax, z10, tWeldGun;
		MoveL [[591.28,-1347.97,82.12],[0.473675,0.523571,-0.526883,0.473181],[-1,-2,3,0],[9E+09,9E+09,9E+09,9E+09,9E+09,9E+09]], vmax, z10, tWeldGun;
		ArcLStart [[589.37,-1365.31,80.43],[0.473686,0.523433,-0.52707,0.473114],[-1,-2,3,0],[9E+09,9E+09,9E+09,9E+09,9E+09,9E+09]], v40, seam13, weld13\Weave:=weave1, fine, tWeldGun;
		ArcLEnd [[622.55,-1366.30,80.01],[0.473684,0.523416,-0.527101,0.4731],[-1,-2,3,0],[9E+09,9E+09,9E+09,9E+09,9E+09,9E+09]], v10, seam13, weld13\Weave:=weave1, fine, tWeldGun;
		MoveL [[621.57,-1338.36,83.93],[0.473691,0.523533,-0.526918,0.473168],[-1,-2,3,0],[9E+09,9E+09,9E+09,9E+09,9E+09,9E+09]], vmax, z10, tWeldGun;
		MoveJ [[584.48,-948.55,-60.93],[0.252385,-0.649774,-0.664987,-0.268121],[-1,0,0,0],[9E+09,9E+09,9E+09,9E+09,9E+09,9E+09]], vmax, z10, tWeldGun;
		MoveL [[587.25,-889.04,-107.33],[0.252799,-0.649451,-0.665162,-0.268079],[-1,0,0,0],[9E+09,9E+09,9E+09,9E+09,9E+09,9E+09]], vmax, z10, tWeldGun;
		ArcLStart [[584.57,-887.97,-132.03],[0.253395,-0.649148,-0.665278,-0.267962],[-1,0,0,0],[9E+09,9E+09,9E+09,9E+09,9E+09,9E+09]], v40, seam13, weld13\Weave:=weave1, fine, tWeldGun;
		ArcL [[579.79,-893.28,-132.83],[0.253299,-0.649198,-0.665271,-0.26795],[-1,0,0,0],[9E+09,9E+09,9E+09,9E+09,9E+09,9E+09]], v10, seam13, weld13\Weave:=weave1, z0, tWeldGun;
		ArcL [[474.14,-892.61,-132.85],[0.253414,-0.649221,-0.665181,-0.268007],[-1,0,0,0],[9E+09,9E+09,9E+09,9E+09,9E+09,9E+09]], v10, seam13, weld13\Weave:=weave1, z0, tWeldGun;
		ArcLEnd [[466.26,-881.37,-133.85],[0.253479,-0.649182,-0.665197,-0.268001],[-1,0,0,0],[9E+09,9E+09,9E+09,9E+09,9E+09,9E+09]], v10, seam13, weld13\Weave:=weave1, fine, tWeldGun;
		MoveL [[472.59,-879.09,-111.98],[0.253025,-0.6494,-0.665124,-0.268085],[-1,0,0,0],[9E+09,9E+09,9E+09,9E+09,9E+09,9E+09]], vmax, z10, tWeldGun;
		MoveL [[396.83,-879.33,-105.08],[0.253072,-0.649383,-0.665131,-0.268064],[-1,0,0,0],[9E+09,9E+09,9E+09,9E+09,9E+09,9E+09]], vmax, z10, tWeldGun;
		ArcLStart [[395.75,-881.23,-133.67],[0.258521,-0.647234,-0.667343,-0.262506],[-1,-1,0,0],[9E+09,9E+09,9E+09,9E+09,9E+09,9E+09]], v40, seam13, weld13\Weave:=weave1, fine, tWeldGun;
		ArcL [[386.24,-892.71,-134.47],[0.258763,-0.647185,-0.667251,-0.262622],[-1,-1,0,0],[9E+09,9E+09,9E+09,9E+09,9E+09,9E+09]], v10, seam13, weld13\Weave:=weave1, z0, tWeldGun;
		ArcLEnd [[340.78,-892.85,-134.30],[0.258675,-0.647186,-0.6673,-0.262583],[-1,0,0,0],[9E+09,9E+09,9E+09,9E+09,9E+09,9E+09]], v10, seam13, weld13\Weave:=weave1, fine, tWeldGun;
		MoveL [[339.41,-899.45,-120.68],[0.253156,-0.64953,-0.664892,-0.26822],[-1,0,0,0],[9E+09,9E+09,9E+09,9E+09,9E+09,9E+09]], vmax, z10, tWeldGun;
		MoveL [[273.41,-894.64,-124.57],[0.25314,-0.649501,-0.664982,-0.268082],[-1,0,0,0],[9E+09,9E+09,9E+09,9E+09,9E+09,9E+09]], vmax, z10, tWeldGun;
		ArcLStart [[273.64,-892.55,-135.89],[0.253143,-0.64948,-0.665008,-0.268066],[-1,0,0,0],[9E+09,9E+09,9E+09,9E+09,9E+09,9E+09]], v40, seam13, weld13\Weave:=weave1, fine, tWeldGun;
		ArcLEnd [[228.37,-892.49,-135.84],[0.253505,-0.649368,-0.6649,-0.268264],[-1,0,0,0],[9E+09,9E+09,9E+09,9E+09,9E+09,9E+09]], v10, seam13, weld13\Weave:=weave1, fine, tWeldGun;
		MoveL [[221.58,-928.39,28.18],[0.253244,-0.649506,-0.664879,-0.268227],[-1,0,0,0],[9E+09,9E+09,9E+09,9E+09,9E+09,9E+09]], vmax, z10, tWeldGun;
		MoveL [[149.11,-928.37,24.70],[0.253259,-0.649498,-0.664878,-0.268235],[-1,0,0,0],[9E+09,9E+09,9E+09,9E+09,9E+09,9E+09]], vmax, z10, tWeldGun;
		MoveL [[162.69,-898.74,-125.22],[0.226585,-0.659714,-0.673956,-0.243353],[-1,0,0,0],[9E+09,9E+09,9E+09,9E+09,9E+09,9E+09]], vmax, z10, tWeldGun;
		ArcLStart [[162.68,-894.34,-134.19],[0.226618,-0.659727,-0.673924,-0.243377],[-1,0,0,0],[9E+09,9E+09,9E+09,9E+09,9E+09,9E+09]], v40, seam13, weld13\Weave:=weave1, fine, tWeldGun;
		ArcL [[145.47,-893.34,-134.20],[0.226617,-0.659728,-0.673926,-0.243369],[-1,0,0,0],[9E+09,9E+09,9E+09,9E+09,9E+09,9E+09]], v10, seam13, weld13\Weave:=weave1, z0, tWeldGun;
		ArcLEnd [[138.08,-883.34,-135.00],[0.226617,-0.659736,-0.673916,-0.243375],[-1,0,0,0],[9E+09,9E+09,9E+09,9E+09,9E+09,9E+09]], v10, seam13, weld13\Weave:=weave1, fine, tWeldGun;
		MoveL [[143.44,-899.06,25.66],[0.226502,-0.659746,-0.673948,-0.243368],[-1,0,0,0],[9E+09,9E+09,9E+09,9E+09,9E+09,9E+09]], vmax, z10, tWeldGun;
		MoveJ [[133.84,-1301.69,-30.86],[0.241723,0.664636,-0.669792,0.226294],[-1,-1,-2,0],[9E+09,9E+09,9E+09,9E+09,9E+09,9E+09]], vmax, z10, tWeldGun;
		MoveL [[128.93,-1364.55,-117.75],[0.241885,0.664518,-0.669816,0.226396],[-1,-1,-2,0],[9E+09,9E+09,9E+09,9E+09,9E+09,9E+09]], vmax, z10, tWeldGun;
		ArcLStart [[130.22,-1362.66,-133.00],[0.241742,0.664656,-0.669795,0.226206],[-1,-1,-2,0],[9E+09,9E+09,9E+09,9E+09,9E+09,9E+09]], v40, seam13, weld13\Weave:=weave1, fine, tWeldGun;
		ArcLEnd [[139.82,-1352.65,-133.00],[0.241741,0.664664,-0.669789,0.226199],[-1,-1,-2,0],[9E+09,9E+09,9E+09,9E+09,9E+09,9E+09]], v10, seam13, weld13\Weave:=weave1, fine, tWeldGun;
		MoveL [[140.84,-1281.82,33.20],[0.241757,0.664658,-0.669788,0.226201],[-1,-1,-2,0],[9E+09,9E+09,9E+09,9E+09,9E+09,9E+09]], vmax, z10, tWeldGun;
		MoveL [[199.15,-1314.71,46.47],[0.241551,0.664904,-0.669698,0.225967],[-1,0,-2,0],[9E+09,9E+09,9E+09,9E+09,9E+09,9E+09]], vmax, z10, tWeldGun;
		MoveL [[198.91,-1343.90,-125.14],[0.241811,0.664705,-0.669734,0.226168],[-1,0,-2,0],[9E+09,9E+09,9E+09,9E+09,9E+09,9E+09]], vmax, z10, tWeldGun;
		ArcLStart [[198.90,-1353.69,-133.34],[0.241812,0.664727,-0.669715,0.226157],[-1,0,-2,0],[9E+09,9E+09,9E+09,9E+09,9E+09,9E+09]], v40, seam13, weld13\Weave:=weave1, fine, tWeldGun;
		ArcLEnd [[273.03,-1353.83,-133.84],[0.241819,0.664737,-0.669703,0.226158],[-1,0,-2,0],[9E+09,9E+09,9E+09,9E+09,9E+09,9E+09]], v10, seam13, weld13\Weave:=weave1, fine, tWeldGun;
		MoveL [[270.78,-1352.99,-112.59],[0.24181,0.664694,-0.669682,0.226354],[-1,0,-2,0],[9E+09,9E+09,9E+09,9E+09,9E+09,9E+09]], vmax, z10, tWeldGun;
		MoveL [[334.63,-1344.14,-112.65],[0.24179,0.664653,-0.669743,0.226317],[-1,0,-2,0],[9E+09,9E+09,9E+09,9E+09,9E+09,9E+09]], vmax, z10, tWeldGun;
		ArcLStart [[334.60,-1355.56,-132.86],[0.241804,0.664676,-0.669714,0.226319],[-1,0,-2,0],[9E+09,9E+09,9E+09,9E+09,9E+09,9E+09]], v40, seam13, weld13\Weave:=weave1, fine, tWeldGun;
		ArcL [[379.61,-1357.00,-133.48],[0.241803,0.664721,-0.66968,0.22629],[-1,0,-2,0],[9E+09,9E+09,9E+09,9E+09,9E+09,9E+09]], v10, seam13, weld13\Weave:=weave1, z0, tWeldGun;
		ArcLEnd [[388.22,-1366.34,-133.46],[0.241795,0.664755,-0.669657,0.226266],[-1,0,-2,0],[9E+09,9E+09,9E+09,9E+09,9E+09,9E+09]], v10, seam13, weld13\Weave:=weave1, fine, tWeldGun;
		MoveL [[388.15,-1371.45,-115.55],[0.241783,0.664794,-0.669629,0.226246],[-1,0,-2,0],[9E+09,9E+09,9E+09,9E+09,9E+09,9E+09]], vmax, z10, tWeldGun;
		MoveL [[460.68,-1363.89,-125.97],[0.241779,0.664811,-0.669612,0.226249],[-1,0,-2,0],[9E+09,9E+09,9E+09,9E+09,9E+09,9E+09]], vmax, z10, tWeldGun;
		ArcLStart [[460.21,-1367.35,-133.41],[0.241778,0.664844,-0.66959,0.226221],[-1,0,-2,0],[9E+09,9E+09,9E+09,9E+09,9E+09,9E+09]], v40, seam13, weld13\Weave:=weave1, fine, tWeldGun;
		ArcL [[471.28,-1356.20,-133.19],[0.241765,0.664907,-0.669535,0.226213],[-1,0,-2,0],[9E+09,9E+09,9E+09,9E+09,9E+09,9E+09]], v10, seam13, weld13\Weave:=weave1, z0, tWeldGun;
		ArcL [[572.11,-1358.43,-132.61],[0.241773,0.664896,-0.669549,0.226194],[-1,0,-2,0],[9E+09,9E+09,9E+09,9E+09,9E+09,9E+09]], v10, seam13, weld13\Weave:=weave1, z0, tWeldGun;
		ArcLEnd [[579.23,-1367.64,-131.03],[0.241775,0.66489,-0.66956,0.226176],[-1,0,-2,0],[9E+09,9E+09,9E+09,9E+09,9E+09,9E+09]], v10, seam13, weld13\Weave:=weave1, fine, tWeldGun;
		MoveL [[580.73,-1359.16,-109.60],[0.211837,0.675037,-0.658293,0.257101],[-1,0,-2,0],[9E+09,9E+09,9E+09,9E+09,9E+09,9E+09]], vmax, z10, tWeldGun;
		MoveL [[580.72,-1333.23,219.73],[0.211837,0.67505,-0.658281,0.257098],[-1,0,-2,0],[9E+09,9E+09,9E+09,9E+09,9E+09,9E+09]], vmax, z10, tWeldGun;
		MoveJ [[285.51,-1411.06,96.42],[0.200981,-0.684372,-0.670688,-0.203517],[-1,-1,0,0],[9E+09,9E+09,9E+09,9E+09,9E+09,9E+09]], vmax, z10, tWeldGun;
		MoveL [[278.82,-1413.93,-119.52],[0.177179,-0.688242,-0.683987,-0.164602],[-1,-1,0,0],[9E+09,9E+09,9E+09,9E+09,9E+09,9E+09]], vmax, z10, tWeldGun;
		ArcLStart [[281.58,-1410.59,-130.76],[0.177219,-0.68822,-0.684004,-0.164578],[-1,-1,0,0],[9E+09,9E+09,9E+09,9E+09,9E+09,9E+09]], v40, seam13, weld13\Weave:=weave1, fine, tWeldGun;
		ArcLEnd [[345.51,-1410.56,-130.43],[0.177233,-0.688193,-0.684033,-0.164557],[-1,-1,0,0],[9E+09,9E+09,9E+09,9E+09,9E+09,9E+09]], v10, seam13, weld13\Weave:=weave1, fine, tWeldGun;
		MoveL [[345.60,-1413.44,-114.91],[0.177186,-0.688241,-0.683983,-0.164611],[-1,-1,0,0],[9E+09,9E+09,9E+09,9E+09,9E+09,9E+09]], vmax, z10, tWeldGun;
		MoveL [[346.28,-1410.71,-125.24],[0.247919,-0.667278,-0.662996,-0.231763],[-1,-1,0,0],[9E+09,9E+09,9E+09,9E+09,9E+09,9E+09]], vmax, z10, tWeldGun;
		ArcLStart [[346.10,-1407.24,-130.88],[0.247984,-0.667276,-0.662981,-0.231741],[-1,-1,0,0],[9E+09,9E+09,9E+09,9E+09,9E+09,9E+09]], v20, seam13, weld13\Weave:=weave1, fine, tWeldGun;
		ArcLEnd [[278.11,-1407.26,-130.90],[0.247977,-0.667291,-0.662967,-0.231744],[-1,-1,0,0],[9E+09,9E+09,9E+09,9E+09,9E+09,9E+09]], v10, seam13, weld13\Weave:=weave1, fine, tWeldGun;
		MoveL [[278.24,-1414.33,-118.08],[0.247841,-0.667243,-0.663091,-0.231675],[-1,-1,0,0],[9E+09,9E+09,9E+09,9E+09,9E+09,9E+09]], vmax, z10, tWeldGun;
		MoveJ [[748.76,-1435.11,122.90],[0.309636,-0.639534,-0.632199,-0.308944],[-1,0,0,0],[9E+09,9E+09,9E+09,9E+09,9E+09,9E+09]], vmax, z10, tWeldGun;
		MoveL [[713.11,-1431.01,114.74],[0.309534,-0.639554,-0.632247,-0.308909],[-1,0,0,0],[9E+09,9E+09,9E+09,9E+09,9E+09,9E+09]], vmax, z10, tWeldGun;
		ArcLStart [[713.04,-1412.89,114.87],[0.309691,-0.63953,-0.632161,-0.308975],[-1,0,0,0],[9E+09,9E+09,9E+09,9E+09,9E+09,9E+09]], v40, seam13, weld13\Weave:=weave1, fine, tWeldGun;
		ArcLEnd [[694.58,-1412.99,89.29],[0.309707,-0.639496,-0.632205,-0.30894],[-1,0,0,0],[9E+09,9E+09,9E+09,9E+09,9E+09,9E+09]], v10, seam13, weld13\Weave:=weave1, fine, tWeldGun;
		MoveL [[694.62,-1427.85,89.22],[0.309609,-0.639506,-0.63227,-0.308883],[-1,0,0,0],[9E+09,9E+09,9E+09,9E+09,9E+09,9E+09]], v10, z10, tWeldGun;
		MoveL [[713.06,-1431.01,114.71],[0.309564,-0.639548,-0.632251,-0.30888],[-1,0,0,0],[9E+09,9E+09,9E+09,9E+09,9E+09,9E+09]], v10, z10, tWeldGun;
		ArcLStart [[713.01,-1412.95,114.83],[0.309674,-0.639526,-0.632181,-0.308961],[-1,0,0,0],[9E+09,9E+09,9E+09,9E+09,9E+09,9E+09]], v10, seam13, weld13\Weave:=weave1, fine, tWeldGun;
		ArcL [[754.36,-1412.19,114.69],[0.309723,-0.639526,-0.632176,-0.308923],[-1,0,0,0],[9E+09,9E+09,9E+09,9E+09,9E+09,9E+09]], v10, seam13, weld13\Weave:=weave1, z20, tWeldGun;
		ArcL [[760.51,-1413.29,95.28],[0.309812,-0.639541,-0.632089,-0.308979],[-1,0,0,0],[9E+09,9E+09,9E+09,9E+09,9E+09,9E+09]], v10, seam13, weld13\Weave:=weave1, z20, tWeldGun;
		ArcLEnd [[773.26,-1412.05,85.51],[0.309836,-0.639558,-0.632055,-0.30899],[-1,0,0,0],[9E+09,9E+09,9E+09,9E+09,9E+09,9E+09]], v10, seam13, weld13\Weave:=weave1, fine, tWeldGun;
		MoveL [[772.20,-1434.22,91.41],[0.309863,-0.63952,-0.632095,-0.30896],[-1,0,0,0],[9E+09,9E+09,9E+09,9E+09,9E+09,9E+09]], vmax, z10, tWeldGun;
		MoveL [[627.48,-1417.65,-2.71],[0.30978,-0.639664,-0.632044,-0.308849],[-1,0,0,0],[9E+09,9E+09,9E+09,9E+09,9E+09,9E+09]], vmax, z10, tWeldGun;
		ArcLStart [[627.90,-1411.38,-7.20],[0.309892,-0.639531,-0.632205,-0.30868],[-1,0,0,0],[9E+09,9E+09,9E+09,9E+09,9E+09,9E+09]], v40, seam13, weld13\Weave:=weave1, fine, tWeldGun;
		ArcL [[591.09,-1409.57,-56.84],[0.309931,-0.639546,-0.632153,-0.308718],[-1,0,0,0],[9E+09,9E+09,9E+09,9E+09,9E+09,9E+09]], v10, seam13, weld13\Weave:=weave1, z0, tWeldGun;
		ArcLEnd [[542.91,-1408.34,-132.78],[0.310062,-0.639544,-0.632098,-0.308705],[-1,0,0,0],[9E+09,9E+09,9E+09,9E+09,9E+09,9E+09]], v10, seam13, weld13\Weave:=weave1, fine, tWeldGun;
		MoveL [[545.98,-1470.65,-122.68],[0.309529,-0.639772,-0.632153,-0.308653],[-1,0,0,0],[9E+09,9E+09,9E+09,9E+09,9E+09,9E+09]], vmax, z10, tWeldGun;
		MoveL [[546.01,-1470.74,261.49],[0.309463,-0.639811,-0.632171,-0.308601],[-1,0,0,0],[9E+09,9E+09,9E+09,9E+09,9E+09,9E+09]], vmax, z10, tWeldGun;
		MoveJ [[450.72,-1393.79,89.08],[0.00680651,0.918501,-0.0118982,0.395183],[-1,0,-3,0],[9E+09,9E+09,9E+09,9E+09,9E+09,9E+09]], vmax, z10, tWeldGun;
		MoveL [[571.40,-1393.78,20.15],[0.00679519,0.918514,-0.0118615,0.395152],[-1,0,-3,0],[9E+09,9E+09,9E+09,9E+09,9E+09,9E+09]], vmax, z10, tWeldGun;
		ArcLStart [[578.12,-1396.98,11.30],[0.00341351,0.944482,-0.011944,0.328329],[-1,-1,-3,0],[9E+09,9E+09,9E+09,9E+09,9E+09,9E+09]], v50, seam13, weld13\Weave:=weave1, fine, tWeldGun;
		ArcLEnd [[576.85,-1373.89,12.01],[0.00333038,0.944494,-0.0119426,0.328296],[-1,-1,-3,0],[9E+09,9E+09,9E+09,9E+09,9E+09,9E+09]], v10, seam13, weld13\Weave:=weave1, fine, tWeldGun;
		MoveL [[564.04,-1375.65,36.36],[0.00687019,0.918524,-0.0118557,0.395129],[-1,0,-3,0],[9E+09,9E+09,9E+09,9E+09,9E+09,9E+09]], vmax, z10, tWeldGun;
		MoveJ [[280.70,-816.60,118.66],[0.243228,0.672922,-0.664156,0.216597],[-1,0,-2,0],[9E+09,9E+09,9E+09,9E+09,9E+09,9E+09]], vmax, z10, tWeldGun;
		MoveL [[280.25,-835.42,-125.82],[0.19707,0.688443,-0.669204,0.198435],[-1,0,-2,0],[9E+09,9E+09,9E+09,9E+09,9E+09,9E+09]], vmax, z10, tWeldGun;
		ArcLStart [[280.30,-837.36,-134.80],[0.197049,0.688448,-0.669224,0.198371],[-1,0,-2,0],[9E+09,9E+09,9E+09,9E+09,9E+09,9E+09]], v40, seam13, weld13\Weave:=weave1, fine, tWeldGun;
		ArcLEnd [[342.48,-837.33,-134.82],[0.197045,0.688456,-0.669221,0.19836],[-1,0,-2,0],[9E+09,9E+09,9E+09,9E+09,9E+09,9E+09]], v10, seam13, weld13\Weave:=weave1, fine, tWeldGun;
		MoveL [[342.48,-807.65,-103.06],[0.243058,0.673116,-0.664102,0.216347],[-1,0,-2,0],[9E+09,9E+09,9E+09,9E+09,9E+09,9E+09]], vmax, z10, tWeldGun;
		MoveL [[344.84,-838.46,-130.27],[0.239446,0.676384,-0.664309,0.209437],[-1,0,-2,0],[9E+09,9E+09,9E+09,9E+09,9E+09,9E+09]], v40, z10, tWeldGun;
		ArcLStart [[344.43,-840.85,-132.67],[0.274188,0.684847,-0.63395,0.232193],[-1,-1,-2,0],[9E+09,9E+09,9E+09,9E+09,9E+09,9E+09]], v20, seam13, weld13\Weave:=weave1, fine, tWeldGun;
		ArcLEnd [[273.43,-840.83,-132.68],[0.274188,0.684851,-0.633948,0.232188],[-1,-1,-2,0],[9E+09,9E+09,9E+09,9E+09,9E+09,9E+09]], v10, seam13, weld13\Weave:=weave1, fine, tWeldGun;
		MoveL [[282.15,-832.82,-127.25],[0.239444,0.676452,-0.664242,0.209434],[-1,0,-2,0],[9E+09,9E+09,9E+09,9E+09,9E+09,9E+09]], vmax, z10, tWeldGun;
		MoveL [[714.08,-820.90,116.19],[0.255079,0.669279,-0.660332,0.225751],[-1,0,-2,0],[9E+09,9E+09,9E+09,9E+09,9E+09,9E+09]], vmax, z10, tWeldGun;
		ArcLStart [[712.61,-838.41,114.78],[0.255091,0.669302,-0.660306,0.225744],[-1,0,-2,0],[9E+09,9E+09,9E+09,9E+09,9E+09,9E+09]], v40, seam13, weld13\Weave:=weave1, fine, tWeldGun;
		ArcLEnd [[693.55,-838.43,87.96],[0.255107,0.669344,-0.660257,0.225745],[-1,0,-2,0],[9E+09,9E+09,9E+09,9E+09,9E+09,9E+09]], v10, seam13, weld13\Weave:=weave1, fine, tWeldGun;
		MoveL [[693.54,-821.10,87.96],[0.255102,0.669397,-0.660268,0.225562],[-1,0,-2,0],[9E+09,9E+09,9E+09,9E+09,9E+09,9E+09]], v10, z10, tWeldGun;
		MoveL [[714.11,-820.85,116.18],[0.255054,0.669249,-0.660379,0.225731],[-1,0,-2,0],[9E+09,9E+09,9E+09,9E+09,9E+09,9E+09]], v10, z10, tWeldGun;
		ArcLStart [[712.62,-838.42,114.78],[0.255121,0.66926,-0.660338,0.225741],[-1,0,-2,0],[9E+09,9E+09,9E+09,9E+09,9E+09,9E+09]], v10, seam13, weld13\Weave:=weave1, fine, tWeldGun;
		ArcL [[756.22,-838.49,114.79],[0.255112,0.669269,-0.660322,0.225772],[-1,0,-2,0],[9E+09,9E+09,9E+09,9E+09,9E+09,9E+09]], v10, seam13, weld13\Weave:=weave1, z10, tWeldGun;
		ArcL [[758.84,-838.47,95.77],[0.255122,0.669244,-0.660353,0.225742],[-1,0,-2,0],[9E+09,9E+09,9E+09,9E+09,9E+09,9E+09]], v10, seam13, weld13\Weave:=weave1, z10, tWeldGun;
		ArcLEnd [[772.06,-838.21,86.77],[0.25512,0.669202,-0.660399,0.225733],[-1,0,-2,0],[9E+09,9E+09,9E+09,9E+09,9E+09,9E+09]], v10, seam13, weld13\Weave:=weave1, fine, tWeldGun;
		MoveL [[772.08,-767.27,86.77],[0.255103,0.66918,-0.660433,0.225721],[-1,0,-2,0],[9E+09,9E+09,9E+09,9E+09,9E+09,9E+09]], vmax, z10, tWeldGun;
		MoveL [[627.18,-826.93,-5.83],[0.253508,0.65756,-0.66005,0.26016],[-1,0,-2,0],[9E+09,9E+09,9E+09,9E+09,9E+09,9E+09]], vmax, z10, tWeldGun;
		ArcLStart [[628.43,-838.84,-7.42],[0.253583,0.657498,-0.659979,0.260424],[-1,0,-2,0],[9E+09,9E+09,9E+09,9E+09,9E+09,9E+09]], v40, seam13, weld13\Weave:=weave1, fine, tWeldGun;
		ArcL [[590.65,-838.63,-62.79],[0.253573,0.657458,-0.660028,0.260409],[-1,0,-2,0],[9E+09,9E+09,9E+09,9E+09,9E+09,9E+09]], v10, seam13, weld13\Weave:=weave1, z0, tWeldGun;
		ArcLEnd [[541.43,-839.57,-132.20],[0.253576,0.657468,-0.660024,0.260391],[-1,0,-2,0],[9E+09,9E+09,9E+09,9E+09,9E+09,9E+09]], v10, seam13, weld13\Weave:=weave1, fine, tWeldGun;
		MoveL [[548.88,-773.40,234.33],[0.243177,0.673515,-0.663846,0.215757],[-1,0,-2,0],[9E+09,9E+09,9E+09,9E+09,9E+09,9E+09]], vmax, z10, tWeldGun;
		MoveJ [[554.61,-845.95,234.31],[0.0125503,-0.913958,0.00705174,-0.405554],[-1,0,-3,0],[9E+09,9E+09,9E+09,9E+09,9E+09,9E+09]], vmax, z10, tWeldGun;
		MoveL [[577.03,-856.78,17.59],[0.00389083,-0.924944,0.010701,-0.379933],[-1,-1,-3,0],[9E+09,9E+09,9E+09,9E+09,9E+09,9E+09]], vmax, z10, tWeldGun;
		ArcLStart [[582.22,-857.18,9.61],[0.00390717,-0.924951,0.0106639,-0.379916],[-1,-1,-3,0],[9E+09,9E+09,9E+09,9E+09,9E+09,9E+09]], v40, seam13, weld13\Weave:=weave1, fine, tWeldGun;
		ArcLEnd [[579.58,-882.17,9.01],[0.00392765,-0.92496,0.0106159,-0.379896],[-1,-1,-3,0],[9E+09,9E+09,9E+09,9E+09,9E+09,9E+09]], v10, seam13, weld13\Weave:=weave1, fine, tWeldGun;
		MoveL [[536.09,-886.10,63.12],[0.0125865,-0.913974,0.00698526,-0.405519],[-1,0,-3,0],[9E+09,9E+09,9E+09,9E+09,9E+09,9E+09]], vmax, z10, tWeldGun;
		MoveJ [[730.00,-817.88,232.84],[0.157166,-0.839072,-0.35904,-0.37729],[-1,0,0,0],[9E+09,9E+09,9E+09,9E+09,9E+09,9E+09]], vmax, z10, tWeldGun;
		MoveL [[549.10,-773.76,241.36],[0.243257,0.673368,-0.663867,0.216061],[-1,0,2,0],[9E+09,9E+09,9E+09,9E+09,9E+09,9E+09]], vmax, z10, tWeldGun;
		MoveJ [[785.08,-1364.00,203.32],[0.00171317,-0.947718,0.00701896,-0.319029],[-1,-1,1,0],[9E+09,9E+09,9E+09,9E+09,9E+09,9E+09]], vmax, z10, tWeldGun;
		MoveL [[803.47,-1368.09,131.07],[0.00412255,-0.937659,0.00608177,-0.347481],[-1,-1,1,0],[9E+09,9E+09,9E+09,9E+09,9E+09,9E+09]], vmax, z10, tWeldGun;
		ArcLStart [[809.38,-1368.68,123.61],[0.00416001,-0.937677,0.00607274,-0.347432],[-1,-1,1,0],[9E+09,9E+09,9E+09,9E+09,9E+09,9E+09]], v40, seam13, weld13\Weave:=weave1, fine, tWeldGun;
		ArcLEnd [[808.86,-1399.08,123.61],[0.00418964,-0.937686,0.00604111,-0.347406],[-1,-1,1,0],[9E+09,9E+09,9E+09,9E+09,9E+09,9E+09]], v10, seam13, weld13\Weave:=weave1, fine, tWeldGun;
		MoveL [[799.72,-1397.77,160.94],[0.00406041,-0.937645,0.00597838,-0.34752],[-1,-1,1,0],[9E+09,9E+09,9E+09,9E+09,9E+09,9E+09]], vmax, z10, tWeldGun;
		MoveJ [[912.45,-910.97,281.24],[0.471963,-0.00834501,-0.88125,-0.0240746],[-1,-1,-1,0],[9E+09,9E+09,9E+09,9E+09,9E+09,9E+09]], vmax, z10, tWeldGun;
		MoveL [[909.26,-887.50,143.89],[0.306131,-0.0105667,-0.951842,-0.0130303],[-1,0,-1,0],[9E+09,9E+09,9E+09,9E+09,9E+09,9E+09]], vmax, z10, tWeldGun;
		ArcLStart [[898.20,-888.74,123.25],[0.30619,-0.0105743,-0.951822,-0.0130813],[-1,0,-1,0],[9E+09,9E+09,9E+09,9E+09,9E+09,9E+09]], v40, seam13, weld13\Weave:=weave1, fine, tWeldGun;
		ArcLEnd [[898.88,-858.30,123.24],[0.30626,-0.0105439,-0.9518,-0.0131118],[-1,0,-1,0],[9E+09,9E+09,9E+09,9E+09,9E+09,9E+09]], v10, seam13, weld13\Weave:=weave1, fine, tWeldGun;
		MoveL [[912.81,-855.15,147.89],[0.30614,-0.0105141,-0.95184,-0.0129908],[-1,0,-1,0],[9E+09,9E+09,9E+09,9E+09,9E+09,9E+09]], vmax, z10, tWeldGun;
		MoveJ [[902.72,-1362.89,137.84],[0.306146,-0.0105253,-0.951838,-0.0129664],[-1,0,-1,0],[9E+09,9E+09,9E+09,9E+09,9E+09,9E+09]], vmax, z10, tWeldGun;
		MoveL [[908.97,-1368.68,133.52],[0.305903,-0.0107467,-0.951921,-0.0124571],[-1,0,-1,0],[9E+09,9E+09,9E+09,9E+09,9E+09,9E+09]], vmax, z10, tWeldGun;
		ArcLStart [[896.49,-1366.33,124.89],[0.305959,-0.0107753,-0.951901,-0.0125936],[-1,0,-1,0],[9E+09,9E+09,9E+09,9E+09,9E+09,9E+09]], v40, seam13, weld13\Weave:=weave1, fine, tWeldGun;
		ArcLEnd [[896.41,-1395.28,124.44],[0.305998,-0.010735,-0.95189,-0.0124647],[-1,0,-1,0],[9E+09,9E+09,9E+09,9E+09,9E+09,9E+09]], v10, seam13, weld13\Weave:=weave1, fine, tWeldGun;
		MoveL [[900.37,-1394.95,165.72],[0.306084,-0.0106333,-0.95186,-0.0127431],[-1,0,-1,0],[9E+09,9E+09,9E+09,9E+09,9E+09,9E+09]], vmax, z10, tWeldGun;
		MoveJ [[778.65,-875.76,193.58],[0.0091964,-0.885136,-0.0131126,-0.465058],[-1,0,1,0],[9E+09,9E+09,9E+09,9E+09,9E+09,9E+09]], vmax, z10, tWeldGun;
		MoveL [[804.53,-888.57,142.41],[0.00795263,-0.941332,-0.0147738,-0.337067],[-1,-1,1,0],[9E+09,9E+09,9E+09,9E+09,9E+09,9E+09]], vmax, z10, tWeldGun;
		ArcLStart [[810.02,-892.12,121.82],[0.0114809,-0.956989,-0.017097,-0.289394],[-1,-1,1,0],[9E+09,9E+09,9E+09,9E+09,9E+09,9E+09]], v40, seam13, weld13\Weave:=weave1, fine, tWeldGun;
		ArcLEnd [[810.40,-860.92,121.44],[0.0115135,-0.956962,-0.0170483,-0.289484],[-1,-1,1,0],[9E+09,9E+09,9E+09,9E+09,9E+09,9E+09]], v10, seam13, weld13\Weave:=weave1, fine, tWeldGun;
		MoveL [[808.29,-857.12,184.20],[0.00793204,-0.941309,-0.0148666,-0.337126],[-1,-1,1,0],[9E+09,9E+09,9E+09,9E+09,9E+09,9E+09]], vmax, z10, tWeldGun;
		MoveJ [[948.68,-756.38,498.60],[0.0965323,0.230115,0.963612,0.0958222],[-1,0,3,0],[9E+09,9E+09,9E+09,9E+09,9E+09,9E+09]], vmax, z10, tWeldGun;
		MoveJ [[-77.16,-639.19,851.16],[0.250005,-0.698591,-0.608804,-0.280759],[-2,-1,4,0],[9E+09,9E+09,9E+09,9E+09,9E+09,9E+09]], vmax, z10, tWeldGun;
	ENDPROC
	PROC rRUNSide1A()
           	rTestPosTop;
		TPWrite "Side 1 A";
		MoveJ pSafeS1, vmax, fine, tWeldGun;
		!Code Goes Here
		MoveJ [[1195.77,967.47,624.34],[0.0211986,-0.292543,0.866333,0.404273],[0,-1,1,1],[9E+09,9E+09,9E+09,9E+09,9E+09,9E+09]], v1000, z20, tWeldGun;
		MoveJ [[1202.08,958.55,27.66],[0.0678226,-0.111826,0.895436,0.425548],[0,-1,0,1],[9E+09,9E+09,9E+09,9E+09,9E+09,9E+09]], v1000, z20, tWeldGun;
		!SingArea\Wrist;
		MoveL [[1208.05,954.10,0.64],[0.135152,-0.0819873,0.912838,0.376484],[0,0,0,1],[9E+09,9E+09,9E+09,9E+09,9E+09,9E+09]], v1000, z5, tWeldGun;
		ArcLStart [[1210.98,966.05,-0.56],[0.136528,-0.0793545,0.919739,0.359366],[0,0,0,1],[9E+09,9E+09,9E+09,9E+09,9E+09,9E+09]], v5, seam13, weld13\Weave:=weave1, fine, tWeldGun;
		ArcLEnd [[1185.23,966.22,-0.52],[0.13656,-0.0793251,0.919732,0.359378],[0,0,0,1],[9E+09,9E+09,9E+09,9E+09,9E+09,9E+09]], v5, seam13, weld13\Weave:=weave1, fine, tWeldGun;
		MoveL [[1180.50,960.73,100.66],[0.067842,-0.111808,0.895423,0.425576],[0,-1,0,1],[9E+09,9E+09,9E+09,9E+09,9E+09,9E+09]], vmax, z0, tWeldGun;
		MoveL [[867.04,1014.85,67.84],[0.0692843,-0.0563275,0.92497,-0.369403],[0,1,-1,1],[9E+09,9E+09,9E+09,9E+09,9E+09,9E+09]], vmax, z0, tWeldGun;
		MoveL [[869.49,1011.42,-5.10],[0.0692967,-0.0563794,0.924948,-0.369448],[0,1,-1,1],[9E+09,9E+09,9E+09,9E+09,9E+09,9E+09]], vmax, z0, tWeldGun;
		ArcLStart [[870.37,1003.45,-5.38],[0.069212,-0.0564575,0.924916,-0.369532],[0,1,-1,1],[9E+09,9E+09,9E+09,9E+09,9E+09,9E+09]], v5, seam13, weld13\Weave:=weave1, fine, tWeldGun;
		ArcLEnd [[898.36,1003.45,-5.41],[0.0692053,-0.0564613,0.924916,-0.369532],[0,1,-1,1],[9E+09,9E+09,9E+09,9E+09,9E+09,9E+09]], v5, seam13, weld13\Weave:=weave1, fine, tWeldGun;
		MoveL [[886.66,1008.91,119.93],[0.0693309,-0.056349,0.924962,-0.369411],[0,1,-1,1],[9E+09,9E+09,9E+09,9E+09,9E+09,9E+09]], vmax, z0, tWeldGun;
		MoveL [[1179.30,1008.46,86.74],[0.107531,-0.15675,0.912414,-0.362448],[0,0,-1,1],[9E+09,9E+09,9E+09,9E+09,9E+09,9E+09]], vmax, z0, tWeldGun;
		MoveL [[1183.28,1011.87,-7.09],[0.107529,-0.156762,0.912406,-0.362464],[0,0,-1,1],[9E+09,9E+09,9E+09,9E+09,9E+09,9E+09]], vmax, z0, tWeldGun;
		ArcLStart [[1183.40,1007.31,-6.41],[0.107451,-0.156818,0.912372,-0.362548],[0,0,-1,1],[9E+09,9E+09,9E+09,9E+09,9E+09,9E+09]], v5, seam13, weld13\Weave:=weave1, fine, tWeldGun;
		ArcLEnd [[1214.51,1006.63,-6.05],[0.107448,-0.156867,0.912356,-0.362566],[0,0,-1,1],[9E+09,9E+09,9E+09,9E+09,9E+09,9E+09]], v5, seam13, weld13\Weave:=weave1, fine, tWeldGun;
		MoveL [[1201.36,1025.64,129.06],[0.213207,-0.193181,0.897428,-0.334435],[0,0,-1,1],[9E+09,9E+09,9E+09,9E+09,9E+09,9E+09]], vmax, z0, tWeldGun;
		MoveJ [[885.83,967.12,146.79],[0.0390937,-0.243498,0.889932,0.383668],[0,-1,0,1],[9E+09,9E+09,9E+09,9E+09,9E+09,9E+09]], vmax, z0, tWeldGun;
		MoveL [[894.90,956.27,69.85],[0.0870766,0.0253294,0.943056,0.320035],[0,0,0,1],[9E+09,9E+09,9E+09,9E+09,9E+09,9E+09]], vmax, z0, tWeldGun;
		MoveL [[897.77,955.06,6.57],[0.0949838,0.0234038,0.90292,0.418528],[0,0,0,1],[9E+09,9E+09,9E+09,9E+09,9E+09,9E+09]], vmax, z0, tWeldGun;
		ArcLStart [[897.42,965.40,-1.05],[0.094937,0.0234293,0.90297,0.41843],[0,0,0,1],[9E+09,9E+09,9E+09,9E+09,9E+09,9E+09]], v5, seam13, weld13\Weave:=weave1, fine, tWeldGun;
		ArcLEnd [[869.42,966.04,-2.12],[0.0928113,0.0262163,0.917312,0.386314],[0,0,0,1],[9E+09,9E+09,9E+09,9E+09,9E+09,9E+09]], v5, seam13, weld13\Weave:=weave1, fine, tWeldGun;
		MoveL [[862.21,949.49,214.06],[0.0424258,-0.242958,0.89504,0.371585],[0,-1,0,1],[9E+09,9E+09,9E+09,9E+09,9E+09,9E+09]], vmax, z0, tWeldGun;
		MoveL [[1197.39,1502.39,137.74],[0.0213351,-0.292247,0.866338,0.404469],[0,-1,0,1],[9E+09,9E+09,9E+09,9E+09,9E+09,9E+09]], vmax, z0, tWeldGun;
		MoveL [[1212.43,1503.61,12.77],[0.123742,-0.0547004,0.912363,0.386381],[0,0,0,1],[9E+09,9E+09,9E+09,9E+09,9E+09,9E+09]], vmax, z0, tWeldGun;
		ArcLStart [[1212.50,1513.76,0.64],[0.123662,-0.0546741,0.912392,0.386342],[0,0,0,1],[9E+09,9E+09,9E+09,9E+09,9E+09,9E+09]], v5, seam13, weld13\Weave:=weave1, fine, tWeldGun;
		ArcLEnd [[1182.49,1513.74,0.65],[0.123662,-0.0546753,0.912391,0.386344],[0,0,0,1],[9E+09,9E+09,9E+09,9E+09,9E+09,9E+09]], v5, seam13, weld13\Weave:=weave1, fine, tWeldGun;
		MoveL [[1181.48,1503.16,158.48],[0.0212657,-0.292228,0.86634,0.404483],[0,-1,0,1],[9E+09,9E+09,9E+09,9E+09,9E+09,9E+09]], vmax, z0, tWeldGun;
		SingArea\Wrist;
		MoveL [[868.25,1555.51,187.44],[0.227112,-0.185081,0.888817,-0.352378],[0,1,-2,1],[9E+09,9E+09,9E+09,9E+09,9E+09,9E+09]], vmax, z0, tWeldGun;
		MoveL [[868.98,1562.79,2.00],[0.0827412,0.288792,-0.895538,0.328277],[0,1,-2,1],[9E+09,9E+09,9E+09,9E+09,9E+09,9E+09]], vmax, z0, tWeldGun;
		ArcLStart [[868.72,1555.60,-8.90],[0.0827336,0.288835,-0.895505,0.32833],[0,1,-2,1],[9E+09,9E+09,9E+09,9E+09,9E+09,9E+09]], v40, seam13, weld13\Weave:=weave1, fine, tWeldGun;
		ArcLEnd [[890.47,1555.25,-8.94],[0.0827473,0.288833,-0.895496,0.328354],[0,1,-2,1],[9E+09,9E+09,9E+09,9E+09,9E+09,9E+09]], v5, seam13, weld13\Weave:=weave1, fine, tWeldGun;
		MoveL [[888.12,1562.49,80.36],[0.227116,-0.185107,0.888791,-0.352426],[0,1,-2,1],[9E+09,9E+09,9E+09,9E+09,9E+09,9E+09]], vmax, z0, tWeldGun;
		MoveL [[1184.50,1555.09,41.59],[0.152145,-0.176338,0.927538,-0.292285],[0,1,-2,1],[9E+09,9E+09,9E+09,9E+09,9E+09,9E+09]], vmax, z0, tWeldGun;
		MoveL [[1177.05,1568.70,-9.93],[0.112232,0.626696,-0.699388,0.32483],[0,1,-3,1],[9E+09,9E+09,9E+09,9E+09,9E+09,9E+09]], vmax, z0, tWeldGun;
		ArcLStart [[1176.96,1560.25,-11.73],[0.112334,0.626692,-0.699393,0.32479],[0,1,-3,1],[9E+09,9E+09,9E+09,9E+09,9E+09,9E+09]], v30, seam13, weld13\Weave:=weave1, fine, tWeldGun;
		ArcLEnd [[1201.35,1560.20,-11.73],[0.112336,0.626692,-0.699391,0.324794],[0,1,-3,1],[9E+09,9E+09,9E+09,9E+09,9E+09,9E+09]], v5, seam13, weld13\Weave:=weave1, fine, tWeldGun;
		MoveL [[1205.97,1566.31,170.25],[0.227077,-0.185152,0.88879,-0.352432],[0,0,-2,1],[9E+09,9E+09,9E+09,9E+09,9E+09,9E+09]], vmax, z0, tWeldGun;
		MoveL [[881.77,1504.38,147.85],[0.0212859,-0.292306,0.866337,0.404431],[0,-1,0,1],[9E+09,9E+09,9E+09,9E+09,9E+09,9E+09]], vmax, z0, tWeldGun;
		MoveL [[883.67,1496.64,-2.08],[0.003736,0.116344,0.927337,0.355663],[0,0,0,1],[9E+09,9E+09,9E+09,9E+09,9E+09,9E+09]], vmax, z0, tWeldGun;
		ArcLStart [[871.33,1509.38,-5.47],[0.0256096,0.12647,0.911101,0.391464],[0,0,0,1],[9E+09,9E+09,9E+09,9E+09,9E+09,9E+09]], v5, seam13, weld13\Weave:=weave1, fine, tWeldGun;
		ArcLEnd [[895.35,1509.73,-5.96],[0.0255803,0.126578,0.91108,0.391481],[0,0,0,1],[9E+09,9E+09,9E+09,9E+09,9E+09,9E+09]], v5, seam13, weld13\Weave:=weave1, fine, tWeldGun;
		MoveL [[865.68,1505.22,88.67],[0.0212437,-0.292287,0.866358,0.404403],[0,-1,0,1],[9E+09,9E+09,9E+09,9E+09,9E+09,9E+09]], vmax, z0, tWeldGun;
		MoveL [[42.29,1547.28,5.42],[0.0930027,-0.145662,0.911404,0.373466],[1,0,0,1],[9E+09,9E+09,9E+09,9E+09,9E+09,9E+09]], vmax, z0, tWeldGun;
		ArcLStart [[44.94,1559.27,-0.33],[0.0928315,-0.145546,0.911432,0.373485],[1,0,0,1],[9E+09,9E+09,9E+09,9E+09,9E+09,9E+09]], v5, seam13, weld13\Weave:=weave1, fine, tWeldGun;
		ArcLEnd [[11.20,1559.22,-0.37],[0.0928406,-0.145479,0.911445,0.373477],[1,0,0,1],[9E+09,9E+09,9E+09,9E+09,9E+09,9E+09]], v5, seam13, weld13\Weave:=weave1, fine, tWeldGun;
		MoveL [[12.10,1550.46,9.38],[0.0929989,-0.14565,0.911414,0.373447],[1,0,0,1],[9E+09,9E+09,9E+09,9E+09,9E+09,9E+09]], vmax, z0, tWeldGun;
		MoveL [[-278.66,1557.62,11.31],[0.104661,-0.181311,0.91043,0.356779],[1,0,0,1],[9E+09,9E+09,9E+09,9E+09,9E+09,9E+09]], vmax, z0, tWeldGun;
		ArcLStart [[-274.74,1562.21,0.51],[0.104631,-0.181272,0.910419,0.356834],[1,0,0,1],[9E+09,9E+09,9E+09,9E+09,9E+09,9E+09]], v5, seam13, weld13\Weave:=weave1, fine, tWeldGun;
		ArcLEnd [[-309.35,1562.22,0.51],[0.104627,-0.181287,0.910416,0.356836],[1,0,0,1],[9E+09,9E+09,9E+09,9E+09,9E+09,9E+09]], v5, seam13, weld13\Weave:=weave1, fine, tWeldGun;
		MoveL [[-319.66,1562.55,534.71],[0.0907184,-0.623281,0.712938,0.30824],[1,0,0,1],[9E+09,9E+09,9E+09,9E+09,9E+09,9E+09]], vmax, z0, tWeldGun;
		MoveJ [[-204.06,743.62,410.35],[0.169831,0.702229,0.669586,-0.1723],[1,0,-2,0],[9E+09,9E+09,9E+09,9E+09,9E+09,9E+09]], vmax, z0, tWeldGun;
		MoveJ [[-336.86,555.26,14.49],[0.352891,0.90921,0.19794,-0.0981131],[0,0,-2,0],[9E+09,9E+09,9E+09,9E+09,9E+09,9E+09]], vmax, z0, tWeldGun;
		ArcLStart [[-339.40,546.11,8.17],[0.352916,0.909193,0.197986,-0.0980848],[0,0,-2,0],[9E+09,9E+09,9E+09,9E+09,9E+09,9E+09]], v5, seam13, weld13\Weave:=weave1, fine, tWeldGun;
		ArcLEnd [[-308.18,546.22,10.17],[0.352965,0.909174,0.197991,-0.0980798],[0,0,-2,0],[9E+09,9E+09,9E+09,9E+09,9E+09,9E+09]], v5, seam13, weld13\Weave:=weave1, fine, tWeldGun;
		MoveL [[-306.62,555.42,20.36],[0.352823,0.909224,0.197986,-0.0981282],[0,0,-2,0],[9E+09,9E+09,9E+09,9E+09,9E+09,9E+09]], vmax, z0, tWeldGun;
		MoveL [[-15.36,553.36,14.76],[0.325268,0.908092,0.244403,-0.0991795],[0,0,-2,0],[9E+09,9E+09,9E+09,9E+09,9E+09,9E+09]], vmax, z0, tWeldGun;
		ArcLStart [[-20.57,543.16,6.91],[0.325282,0.908085,0.244435,-0.0991218],[0,0,-2,0],[9E+09,9E+09,9E+09,9E+09,9E+09,9E+09]], v5, seam13, weld13\Weave:=weave1, fine, tWeldGun;
		ArcLEnd [[12.25,543.14,6.91],[0.325307,0.908076,0.24444,-0.0991132],[0,0,-2,0],[9E+09,9E+09,9E+09,9E+09,9E+09,9E+09]], v5, seam13, weld13\Weave:=weave1, fine, tWeldGun;
		MoveL [[16.53,551.56,14.73],[0.325268,0.908096,0.244389,-0.0991872],[0,0,-2,0],[9E+09,9E+09,9E+09,9E+09,9E+09,9E+09]], vmax, z0, tWeldGun;
		MoveL [[835.19,546.59,8.86],[0.354374,0.887507,0.294518,0.00309851],[0,-1,-2,0],[9E+09,9E+09,9E+09,9E+09,9E+09,9E+09]], vmax, z0, tWeldGun;
		ArcLStart [[833.78,537.04,2.86],[0.35438,0.887508,0.29451,0.00299066],[0,-1,-2,0],[9E+09,9E+09,9E+09,9E+09,9E+09,9E+09]], v5, seam13, weld13\Weave:=weave1, fine, tWeldGun;
		ArcLEnd [[865.17,537.05,2.84],[0.354381,0.887511,0.294501,0.00299003],[0,-1,-2,0],[9E+09,9E+09,9E+09,9E+09,9E+09,9E+09]], v5, seam13, weld13\Weave:=weave1, fine, tWeldGun;
		MoveL [[863.15,544.60,13.06],[0.354372,0.887507,0.29452,0.00310136],[0,-1,-2,0],[9E+09,9E+09,9E+09,9E+09,9E+09,9E+09]], vmax, z0, tWeldGun;
		ConfL\Off;
		MoveL [[1163.05,540.25,17.31],[0.272611,0.697866,0.657915,-0.0762502],[0,-1,-3,0],[9E+09,9E+09,9E+09,9E+09,9E+09,9E+09]], vmax, z0, tWeldGun;
		ArcLStart [[1164.07,531.66,5.73],[0.272616,0.697855,0.657924,-0.0762578],[0,-1,-3,0],[9E+09,9E+09,9E+09,9E+09,9E+09,9E+09]], v5, seam13, weld13\Weave:=weave1, fine, tWeldGun;
		ArcLEnd [[1197.06,532.11,5.95],[0.272632,0.697842,0.65793,-0.076274],[0,-1,-3,0],[9E+09,9E+09,9E+09,9E+09,9E+09,9E+09]], v5, seam13, weld13\Weave:=weave1, fine, tWeldGun;
		MoveL [[1196.79,537.72,478.96],[0.266966,0.671404,0.686159,-0.0844522],[0,-1,-3,0],[9E+09,9E+09,9E+09,9E+09,9E+09,9E+09]], vmax, z10, tWeldGun;
		!MoveJ [[44.07,948.69,1172.83],[0.0459633,-0.688402,0.722614,0.0426485],[0,-1,0,0],[9E+09,9E+09,9E+09,9E+09,9E+09,9E+09]], vmax, z10, tWeldGun;
		MoveJ [[-340.94,933.57,290.70],[0.111592,-0.946666,-0.184924,-0.23911],[1,0,-2,0],[9E+09,9E+09,9E+09,9E+09,9E+09,9E+09]], vmax, z10, tWeldGun;
		MoveL [[-397.78,986.25,11.78],[0.351596,0.0366706,-0.934077,-0.0503611],[1,-1,-3,0],[9E+09,9E+09,9E+09,9E+09,9E+09,9E+09]], v1000, z1, tWeldGun;
		ArcLStart [[-402.72,985.80,-7.72],[0.351569,0.0366513,-0.934094,-0.0502539],[1,-1,-3,0],[9E+09,9E+09,9E+09,9E+09,9E+09,9E+09]], v5, seam13, weld13\Weave:=weave1, fine, tWeldGun;
		ArcL [[-401.70,963.07,-8.24],[0.351611,0.0366522,-0.934073,-0.0503387],[1,-1,-3,0],[9E+09,9E+09,9E+09,9E+09,9E+09,9E+09]], v5, seam13, weld13\Weave:=weave1, z1, tWeldGun;
		ArcLEnd [[-423.62,948.43,-7.98],[0.166188,-0.662072,-0.696074,-0.222538],[1,0,-2,0],[9E+09,9E+09,9E+09,9E+09,9E+09,9E+09]], v5, seam13, weld13\Weave:=weave1, fine, tWeldGun;
		MoveL [[-432.50,895.49,94.61],[0.171308,-0.660838,-0.695601,-0.2238],[1,0,-2,0],[9E+09,9E+09,9E+09,9E+09,9E+09,9E+09]], vmax, z0, tWeldGun;
		MoveL [[-428.23,950.42,262.61],[0.171376,-0.660832,-0.695567,-0.223872],[1,0,2,0],[9E+09,9E+09,9E+09,9E+09,9E+09,9E+09]], vmax, z0, tWeldGun;
		MoveJ [[-1240.64,940.49,246.51],[0.200371,-0.594607,-0.764476,-0.147887],[1,0,2,0],[9E+09,9E+09,9E+09,9E+09,9E+09,9E+09]], vmax, z0, tWeldGun;
		MoveL [[-1259.54,939.02,-1.77],[0.21012,-0.673416,-0.681865,-0.193445],[1,0,2,0],[9E+09,9E+09,9E+09,9E+09,9E+09,9E+09]], v100, z0, tWeldGun;
		ArcLStart [[-1260.54,944.62,-7.18],[0.210122,-0.673414,-0.681866,-0.193447],[1,0,2,0],[9E+09,9E+09,9E+09,9E+09,9E+09,9E+09]], v5, seam13, weld13\Weave:=weave1, fine, tWeldGun;
		ArcL [[-1288.12,948.59,-6.58],[0.116094,0.902256,0.096617,0.403884],[1,0,3,0],[9E+09,9E+09,9E+09,9E+09,9E+09,9E+09]], v5, seam13, weld13\Weave:=weave1, z1, tWeldGun;
		ArcLEnd [[-1288.16,971.46,-7.79],[0.116108,0.902247,0.096586,0.403907],[1,0,3,0],[9E+09,9E+09,9E+09,9E+09,9E+09,9E+09]], v5, seam13, weld13\Weave:=weave1, fine, tWeldGun;
		MoveL [[-1282.96,979.96,80.63],[0.116018,0.902243,0.096661,0.403925],[1,0,3,0],[9E+09,9E+09,9E+09,9E+09,9E+09,9E+09]], vmax, z0, tWeldGun;
		MoveJ [[-1358.53,1155.99,133.80],[0.133739,0.955506,0.10811,0.239657],[1,0,3,0],[9E+09,9E+09,9E+09,9E+09,9E+09,9E+09]], vmax, z0, tWeldGun;
		MoveL [[-1362.74,1158.80,0.21],[0.0670489,0.939872,-0.00304011,0.334868],[1,0,3,0],[9E+09,9E+09,9E+09,9E+09,9E+09,9E+09]], vmax, z0, tWeldGun;
		ArcLStart [[-1355.25,1155.18,-6.81],[0.0670685,0.939893,-0.00305685,0.334804],[1,0,3,0],[9E+09,9E+09,9E+09,9E+09,9E+09,9E+09]], v5, seam13, weld13\Weave:=weave1, fine, tWeldGun;
		ArcL [[-1355.69,1177.78,-7.43],[0.0671059,0.939848,-0.00299162,0.334925],[1,0,3,0],[9E+09,9E+09,9E+09,9E+09,9E+09,9E+09]], v5, seam13, weld13\Weave:=weave1, z1, tWeldGun;
		ArcLEnd [[-1334.42,1192.37,-6.00],[0.222223,0.801405,-0.520282,0.194098],[1,0,4,0],[9E+09,9E+09,9E+09,9E+09,9E+09,9E+09]], v5, seam13, weld13\Weave:=weave1, fine, tWeldGun;
		MoveL [[-1328.99,1198.21,13.92],[0.263465,0.723639,-0.589044,0.244868],[1,0,4,0],[9E+09,9E+09,9E+09,9E+09,9E+09,9E+09]], v100, z0, tWeldGun;
		MoveL [[-1329.56,1242.98,151.23],[0.276586,0.758563,-0.567487,0.161373],[1,0,4,0],[9E+09,9E+09,9E+09,9E+09,9E+09,9E+09]], vmax, z0, tWeldGun;
		MoveJ [[-495.18,1248.58,261.21],[0.287177,0.742929,-0.58422,0.155801],[1,0,-1,0],[9E+09,9E+09,9E+09,9E+09,9E+09,9E+09]], vmax, z0, tWeldGun;
		MoveL [[-498.43,1204.30,4.59],[0.287207,0.742912,-0.584227,0.155798],[1,0,-1,0],[9E+09,9E+09,9E+09,9E+09,9E+09,9E+09]], vmax, z0, tWeldGun;
		ArcLStart [[-498.40,1197.60,-6.80],[0.287196,0.742928,-0.584205,0.155827],[1,0,-1,0],[9E+09,9E+09,9E+09,9E+09,9E+09,9E+09]], v5, seam13, weld13\Weave:=weave1, fine, tWeldGun;
		ArcL [[-476.82,1197.38,-9.61],[0.21297,0.671228,-0.679729,0.205102],[1,-1,0,0],[9E+09,9E+09,9E+09,9E+09,9E+09,9E+09]], v5, seam13, weld13\Weave:=weave1, z1, tWeldGun;
		SingArea\Wrist;
		ArcLEnd [[-463.85,1168.99,-9.51],[0.359552,0.0381067,-0.931211,-0.0460231],[1,-1,1,0],[9E+09,9E+09,9E+09,9E+09,9E+09,9E+09]], v5, seam13, weld13\Weave:=weave1, fine, tWeldGun;
		MoveL [[-421.44,1139.09,130.73],[0.359544,0.0381675,-0.931204,-0.0461746],[1,-1,1,0],[9E+09,9E+09,9E+09,9E+09,9E+09,9E+09]], vmax, z0, tWeldGun;
		MoveJ [[-450.31,718.78,85.28],[0.233736,0.658742,-0.674881,0.236565],[1,-1,0,0],[9E+09,9E+09,9E+09,9E+09,9E+09,9E+09]], vmax, z0, tWeldGun;
		MoveL [[-441.01,718.90,-5.39],[0.233736,0.658734,-0.674888,0.236568],[1,-1,0,0],[9E+09,9E+09,9E+09,9E+09,9E+09,9E+09]], vmax, z0, tWeldGun;
		ArcLStart [[-436.93,709.93,-6.17],[0.103288,0.786716,-0.48105,0.372828],[1,-1,0,0],[9E+09,9E+09,9E+09,9E+09,9E+09,9E+09]], v5, seam13, weld13\Weave:=weave1, fine, tWeldGun;
		ArcLEnd [[-412.32,709.94,-7.38],[0.103283,0.786716,-0.481044,0.372837],[1,-1,0,0],[9E+09,9E+09,9E+09,9E+09,9E+09,9E+09]], v5, seam13, weld13\Weave:=weave1, fine, tWeldGun;
		MoveL [[-432.17,783.45,96.50],[0.233754,0.658736,-0.674882,0.23656],[1,-1,0,0],[9E+09,9E+09,9E+09,9E+09,9E+09,9E+09]], vmax, z0, tWeldGun;
		MoveL [[-1257.57,713.89,96.49],[0.233748,0.658741,-0.67488,0.236557],[1,-1,0,0],[9E+09,9E+09,9E+09,9E+09,9E+09,9E+09]], vmax, z0, tWeldGun;
		MoveL [[-1261.90,718.36,0.85],[0.233781,0.658746,-0.674869,0.236543],[1,-1,0,0],[9E+09,9E+09,9E+09,9E+09,9E+09,9E+09]], vmax, z0, tWeldGun;
		ArcLStart [[-1261.47,715.84,-1.13],[0.205901,0.66876,-0.682611,0.210729],[1,-1,0,0],[9E+09,9E+09,9E+09,9E+09,9E+09,9E+09]], v5, seam13, weld13\Weave:=weave1, fine, tWeldGun;
		ArcL [[-1281.65,715.74,-1.11],[0.205892,0.668784,-0.682593,0.210724],[1,-1,0,0],[9E+09,9E+09,9E+09,9E+09,9E+09,9E+09]], v5, seam13, weld13\Weave:=weave1, z1, tWeldGun;
		ArcLEnd [[-1294.10,678.20,-5.73],[0.00242996,-0.947951,0.0663235,-0.311424],[1,0,-1,0],[9E+09,9E+09,9E+09,9E+09,9E+09,9E+09]], v5, seam13, weld13\Weave:=weave1, fine, tWeldGun;
		MoveL [[-1282.90,713.31,123.57],[0.233803,0.658736,-0.674861,0.236572],[1,-1,0,0],[9E+09,9E+09,9E+09,9E+09,9E+09,9E+09]], vmax, z0, tWeldGun;
		MoveJ [[-1344.23,1422.02,101.83],[0.226991,-0.675391,-0.661326,-0.234461],[1,0,-2,0],[9E+09,9E+09,9E+09,9E+09,9E+09,9E+09]], vmax, z0, tWeldGun;
		MoveL [[-1321.45,1421.99,-3.60],[0.227001,-0.67541,-0.661307,-0.234449],[1,0,-2,0],[9E+09,9E+09,9E+09,9E+09,9E+09,9E+09]], vmax, z0, tWeldGun;
		ArcLStart [[-1319.04,1427.22,-11.49],[0.227017,-0.675406,-0.661308,-0.234441],[1,0,-2,0],[9E+09,9E+09,9E+09,9E+09,9E+09,9E+09]], v5, seam13, weld13\Weave:=weave1, fine, tWeldGun;
		ArcL [[-1343.46,1427.11,-9.28],[0.22703,-0.675416,-0.661296,-0.234433],[1,0,-2,0],[9E+09,9E+09,9E+09,9E+09,9E+09,9E+09]], v5, seam13, weld13\Weave:=weave1, z1, tWeldGun;
		ArcLEnd [[-1359.95,1461.83,-9.85],[0.0686283,-0.96088,0.0174311,-0.267764],[1,0,-1,0],[9E+09,9E+09,9E+09,9E+09,9E+09,9E+09]], v5, seam13, weld13\Weave:=weave1, fine, tWeldGun;
		MoveL [[-1320.89,1427.11,81.12],[0.226982,-0.675417,-0.661301,-0.234462],[1,0,-2,0],[9E+09,9E+09,9E+09,9E+09,9E+09,9E+09]], vmax, z0, tWeldGun;
		MoveL [[-494.97,1419.41,70.78],[0.226989,-0.675424,-0.661294,-0.234454],[1,0,-2,0],[9E+09,9E+09,9E+09,9E+09,9E+09,9E+09]], vmax, z0, tWeldGun;
		MoveL [[-494.98,1419.41,-5.90],[0.226987,-0.675436,-0.661284,-0.23445],[1,0,-2,0],[9E+09,9E+09,9E+09,9E+09,9E+09,9E+09]], vmax, z0, tWeldGun;
		ArcLStart [[-493.82,1428.87,-10.09],[0.226985,-0.675462,-0.66126,-0.234445],[1,0,-2,0],[9E+09,9E+09,9E+09,9E+09,9E+09,9E+09]], v5, seam13, weld13\Weave:=weave1, fine, tWeldGun;
		ArcL [[-470.48,1427.72,-10.70],[0.226989,-0.675489,-0.66123,-0.234449],[1,0,-2,0],[9E+09,9E+09,9E+09,9E+09,9E+09,9E+09]], v5, seam13, weld13\Weave:=weave1, z1, tWeldGun;
		ArcLEnd [[-460.41,1465.43,-11.27],[0.383623,-0.0667326,-0.920144,0.041429],[1,0,-3,0],[9E+09,9E+09,9E+09,9E+09,9E+09,9E+09]], v5, seam13, weld13\Weave:=weave1, fine, tWeldGun;
		MoveL [[-196.11,1086.38,621.33],[0.226996,-0.675454,-0.661218,-0.234578],[1,0,-2,0],[9E+09,9E+09,9E+09,9E+09,9E+09,9E+09]], vmax, z0, tWeldGun;

		!code ends here

        MoveJ pSafeS1, vmax, z10, tWeldGun;
	ENDPROC


	PROC longwelds()
		MoveJ [[-537.74,1528.93,225.26],[0.133056,-0.223334,0.96556,0.0105691],[1,-1,1,0],[9E+09,9E+09,9E+09,9E+09,9E+09,9E+09]], v1000, z50, tWeldGun;
		MoveJ [[-534.17,1676.79,-7.31],[0.13306,-0.223351,0.965556,0.0105536],[1,-1,1,0],[9E+09,9E+09,9E+09,9E+09,9E+09,9E+09]], v1000, z50, tWeldGun;
		ArcLStart [[-534.18,1676.79,-10.95],[0.13306,-0.223361,0.965554,0.0105477],[1,-1,1,0],[9E+09,9E+09,9E+09,9E+09,9E+09,9E+09]], v30, seam13, weld13, fine, tWeldGun;
		ArcL [[-544.58,1676.80,-10.94],[0.133063,-0.223367,0.965552,0.0105509],[1,-1,1,0],[9E+09,9E+09,9E+09,9E+09,9E+09,9E+09]], v30, seam13, weld13, z10, tWeldGun;
		ArcL [[-560.58,1676.80,-10.94],[0.133064,-0.223373,0.96555,0.0105523],[1,-1,1,0],[9E+09,9E+09,9E+09,9E+09,9E+09,9E+09]], v30, seam13, weld13, z10, tWeldGun;
		ArcLEnd [[-573.39,1676.78,-10.94],[0.133047,-0.223358,0.965556,0.0105449],[1,-1,1,0],[9E+09,9E+09,9E+09,9E+09,9E+09,9E+09]], v30, seam13, weld13, fine, tWeldGun;
		MoveL [[-573.40,1676.83,-5.98],[0.133038,-0.223382,0.965552,0.0105696],[1,-1,1,0],[9E+09,9E+09,9E+09,9E+09,9E+09,9E+09]], v50, z1, tWeldGun;
		MoveL [[-575.35,1723.62,-6.01],[0.133042,-0.223378,0.965552,0.0105594],[1,-1,1,0],[9E+09,9E+09,9E+09,9E+09,9E+09,9E+09]], v50, z1, tWeldGun;
		ArcLStart [[-575.34,1723.62,-15.03],[0.133047,-0.22338,0.965551,0.0105632],[1,-1,1,0],[9E+09,9E+09,9E+09,9E+09,9E+09,9E+09]], v30, seam13, weld13, fine, tWeldGun;
		ArcL [[-575.34,1697.62,-15.03],[0.133047,-0.22338,0.965551,0.0105669],[1,-1,1,0],[9E+09,9E+09,9E+09,9E+09,9E+09,9E+09]], v30, seam13, weld13, fine, tWeldGun;
		ArcL [[-575.35,1676.62,-15.02],[0.133043,-0.223381,0.965552,0.0105654],[1,-1,1,0],[9E+09,9E+09,9E+09,9E+09,9E+09,9E+09]], v30, seam13, weld13, fine, tWeldGun;
		ArcL [[-575.35,1655.62,-15.02],[0.13304,-0.223383,0.965551,0.010569],[1,-1,1,0],[9E+09,9E+09,9E+09,9E+09,9E+09,9E+09]], v30, seam13, weld13, fine, tWeldGun;
		ArcL [[-575.35,1632.62,-15.03],[0.133037,-0.22338,0.965553,0.0105659],[1,-1,1,0],[9E+09,9E+09,9E+09,9E+09,9E+09,9E+09]], v30, seam13, weld13, fine, tWeldGun;
		ArcLEnd [[-575.35,1606.61,-15.03],[0.133037,-0.223381,0.965552,0.0105613],[1,-1,1,0],[9E+09,9E+09,9E+09,9E+09,9E+09,9E+09]], v30, seam13, weld13, fine, tWeldGun;
		MoveL [[-575.35,1606.60,-1.09],[0.13303,-0.223389,0.965551,0.0105647],[1,-1,1,0],[9E+09,9E+09,9E+09,9E+09,9E+09,9E+09]], v50, z1, tWeldGun;
		MoveL [[-575.34,1585.59,-1.13],[0.133025,-0.223396,0.965551,0.0105485],[1,-1,1,0],[9E+09,9E+09,9E+09,9E+09,9E+09,9E+09]], v50, z1, tWeldGun;
		ArcLStart [[-574.36,1584.60,-16.12],[0.133023,-0.223401,0.96555,0.010553],[1,-1,1,0],[9E+09,9E+09,9E+09,9E+09,9E+09,9E+09]], v30, seam13, weld13\Weave:=weave1, fine, tWeldGun;
		ArcL [[-574.36,1575.59,-16.13],[0.13302,-0.2234,0.96555,0.0105496],[1,-1,1,0],[9E+09,9E+09,9E+09,9E+09,9E+09,9E+09]], v30, seam13, weld13\Weave:=weave1, fine, tWeldGun;
		ArcL [[-573.36,1542.60,-16.12],[0.133024,-0.223405,0.965549,0.0105554],[1,-1,1,0],[9E+09,9E+09,9E+09,9E+09,9E+09,9E+09]], v30, seam13, weld13\Weave:=weave1, fine, tWeldGun;
		ArcL [[-573.37,1523.59,-16.12],[0.133018,-0.223399,0.965551,0.010556],[1,-1,1,0],[9E+09,9E+09,9E+09,9E+09,9E+09,9E+09]], v30, seam13, weld13\Weave:=weave1, fine, tWeldGun;
		ArcLEnd [[-573.36,1500.60,-16.12],[0.133023,-0.223402,0.965549,0.0105616],[1,-1,1,0],[9E+09,9E+09,9E+09,9E+09,9E+09,9E+09]], v30, seam13, weld13\Weave:=weave1, fine, tWeldGun;
		MoveL [[-573.39,1500.62,-2.23],[0.132981,-0.22343,0.965549,0.0105695],[1,-1,1,0],[9E+09,9E+09,9E+09,9E+09,9E+09,9E+09]], v50, z1, tWeldGun;
		MoveL [[-573.39,1485.63,-2.25],[0.132987,-0.223446,0.965544,0.0105683],[1,-1,1,0],[9E+09,9E+09,9E+09,9E+09,9E+09,9E+09]], v50, z1, tWeldGun;
		ArcLStart [[-573.39,1485.63,-15.25],[0.132986,-0.223448,0.965544,0.0105658],[1,-1,1,0],[9E+09,9E+09,9E+09,9E+09,9E+09,9E+09]], v30, seam13, weld13\Weave:=weave1, fine, tWeldGun;
		ArcL [[-573.40,1464.62,-15.25],[0.132977,-0.223444,0.965546,0.0105643],[1,-1,1,0],[9E+09,9E+09,9E+09,9E+09,9E+09,9E+09]], v30, seam13, weld13\Weave:=weave1, fine, tWeldGun;
		ArcL [[-574.40,1445.63,-15.24],[0.132983,-0.223455,0.965542,0.0105677],[1,-1,1,0],[9E+09,9E+09,9E+09,9E+09,9E+09,9E+09]], v30, seam13, weld13\Weave:=weave1, fine, tWeldGun;
		ArcL [[-574.40,1425.64,-15.24],[0.132985,-0.223457,0.965542,0.0105723],[1,-1,1,0],[9E+09,9E+09,9E+09,9E+09,9E+09,9E+09]], v30, seam13, weld13\Weave:=weave1, fine, tWeldGun;
		ArcL [[-574.40,1404.65,-15.23],[0.132998,-0.223476,0.965536,0.0105691],[1,-1,1,0],[9E+09,9E+09,9E+09,9E+09,9E+09,9E+09]], v30, seam13, weld13\Weave:=weave1, fine, tWeldGun;
		ArcL [[-574.41,1387.63,-15.25],[0.132976,-0.223459,0.965543,0.0105667],[1,-1,1,0],[9E+09,9E+09,9E+09,9E+09,9E+09,9E+09]], v30, seam13, weld13\Weave:=weave1, fine, tWeldGun;
		ArcL [[-574.41,1369.63,-15.25],[0.132976,-0.22346,0.965542,0.0105621],[1,-1,1,0],[9E+09,9E+09,9E+09,9E+09,9E+09,9E+09]], v30, seam13, weld13\Weave:=weave1, fine, tWeldGun;
		ArcL [[-574.42,1347.62,-15.25],[0.132967,-0.223444,0.965547,0.0105695],[1,-1,1,0],[9E+09,9E+09,9E+09,9E+09,9E+09,9E+09]], v30, seam13, weld13\Weave:=weave1, fine, tWeldGun;
		ArcL [[-574.42,1329.62,-15.25],[0.132967,-0.223451,0.965546,0.0105668],[1,-1,1,0],[9E+09,9E+09,9E+09,9E+09,9E+09,9E+09]], v30, seam13, weld13\Weave:=weave1, fine, tWeldGun;
		ArcLEnd [[-575.42,1299.63,-13.24],[0.132972,-0.22346,0.965543,0.0105669],[1,-1,1,0],[9E+09,9E+09,9E+09,9E+09,9E+09,9E+09]], v30, seam13, weld13\Weave:=weave1, fine, tWeldGun;
		MoveL [[-575.42,1299.62,3.76],[0.132974,-0.223461,0.965542,0.0105603],[1,-1,1,0],[9E+09,9E+09,9E+09,9E+09,9E+09,9E+09]], v50, z1, tWeldGun;
		MoveL [[-575.41,1292.59,3.73],[0.13296,-0.223451,0.965547,0.0105324],[1,-1,1,0],[9E+09,9E+09,9E+09,9E+09,9E+09,9E+09]], v50, z1, tWeldGun;
		ArcLStart [[-576.42,1292.61,-13.26],[0.132961,-0.223463,0.965544,0.0105395],[1,-1,1,0],[9E+09,9E+09,9E+09,9E+09,9E+09,9E+09]], v30, seam13, weld13\Weave:=weave1, fine, tWeldGun;
		ArcLEnd [[-576.42,1112.60,-13.27],[0.132955,-0.223454,0.965547,0.010535],[1,-1,1,0],[9E+09,9E+09,9E+09,9E+09,9E+09,9E+09]], v30, seam13, weld13\Weave:=weave1, fine, tWeldGun;
		MoveL [[-576.42,1112.59,8.73],[0.132953,-0.22345,0.965548,0.0105277],[1,-1,1,0],[9E+09,9E+09,9E+09,9E+09,9E+09,9E+09]], v30, z1, tWeldGun;
		!MoveL [[-566.80,1587.36,103.77],[0.148014,0.588799,-0.740551,-0.288083],[1,-2,2,0],[9E+09,9E+09,9E+09,9E+09,9E+09,9E+09]], v30, z1, tWeldGun;
		!MoveL [[-566.80,1587.36,103.77],[0.148015,0.588798,-0.740552,-0.288083],[1,-2,2,0],[9E+09,9E+09,9E+09,9E+09,9E+09,9E+09]], v30, z1, tWeldGun;
		MoveJ [[-551.33,863.77,510.66],[0.15147,0.30253,-0.907678,-0.248302],[1,-1,1,0],[9E+09,9E+09,9E+09,9E+09,9E+09,9E+09]], vmax, z1, tWeldGun;
		MoveJ [[-551.34,773.91,9.99],[0.257685,0.331587,-0.885768,-0.197646],[1,-2,2,0],[9E+09,9E+09,9E+09,9E+09,9E+09,9E+09]], vmax, z1, tWeldGun;
		MoveL [[-569.03,771.59,1.41],[0.257705,0.331593,-0.885761,-0.197643],[1,-2,2,0],[9E+09,9E+09,9E+09,9E+09,9E+09,9E+09]], vmax, z1, tWeldGun;
		ArcLStart [[-569.03,771.58,-13.78],[0.257704,0.331613,-0.885754,-0.197643],[1,-2,2,0],[9E+09,9E+09,9E+09,9E+09,9E+09,9E+09]], v50, seam13, weld13\Weave:=weave1, fine, tWeldGun;
		ArcLEnd [[-568.49,798.58,-13.77],[0.257712,0.331608,-0.885753,-0.197645],[1,-2,2,0],[9E+09,9E+09,9E+09,9E+09,9E+09,9E+09]], v50, seam13, weld13\Weave:=weave1, fine, tWeldGun;
		MoveL [[-568.49,798.57,-7.98],[0.257716,0.331598,-0.885756,-0.197639],[1,-2,2,0],[9E+09,9E+09,9E+09,9E+09,9E+09,9E+09]], vmax, z1, tWeldGun;
		MoveL [[-567.50,823.73,-8.00],[0.257718,0.33163,-0.885749,-0.197615],[1,-2,2,0],[9E+09,9E+09,9E+09,9E+09,9E+09,9E+09]], vmax, z1, tWeldGun;
		ArcLStart [[-569.72,823.72,-13.19],[0.25773,0.331648,-0.88574,-0.197612],[1,-2,2,0],[9E+09,9E+09,9E+09,9E+09,9E+09,9E+09]], v50, seam13, weld13\Weave:=weave1, fine, tWeldGun;
		ArcLEnd [[-568.63,850.44,-13.40],[0.257728,0.331633,-0.885747,-0.197607],[1,-2,2,0],[9E+09,9E+09,9E+09,9E+09,9E+09,9E+09]], v50, seam13, weld13\Weave:=weave1, fine, tWeldGun;
		MoveL [[-568.64,850.44,-6.99],[0.257739,0.331614,-0.88575,-0.197611],[1,-2,2,0],[9E+09,9E+09,9E+09,9E+09,9E+09,9E+09]], vmax, z1, tWeldGun;
		MoveL [[-567.78,877.79,-7.01],[0.257734,0.331631,-0.885748,-0.1976],[1,-2,2,0],[9E+09,9E+09,9E+09,9E+09,9E+09,9E+09]], vmax, z1, tWeldGun;
		ArcLStart [[-568.78,876.58,-13.99],[0.257742,0.331637,-0.885742,-0.197602],[1,-2,2,0],[9E+09,9E+09,9E+09,9E+09,9E+09,9E+09]], v40, seam13, weld13\Weave:=weave1, fine, tWeldGun;
		ArcLEnd [[-569.59,895.98,-14.18],[0.257742,0.331687,-0.885727,-0.197589],[1,-2,2,0],[9E+09,9E+09,9E+09,9E+09,9E+09,9E+09]], v40, seam13, weld13\Weave:=weave1, fine, tWeldGun;
		MoveL [[-569.52,896.01,-8.19],[0.257699,0.331627,-0.885753,-0.197628],[1,-2,2,0],[9E+09,9E+09,9E+09,9E+09,9E+09,9E+09]], vmax, z1, tWeldGun;
		MoveL [[-569.26,927.41,-8.18],[0.257701,0.331632,-0.885751,-0.197629],[1,-2,2,0],[9E+09,9E+09,9E+09,9E+09,9E+09,9E+09]], vmax, z1, tWeldGun;
		ArcLStart [[-569.27,927.40,-14.18],[0.257703,0.331665,-0.88574,-0.197617],[1,-2,2,0],[9E+09,9E+09,9E+09,9E+09,9E+09,9E+09]], v40, seam13, weld13\Weave:=weave1, fine, tWeldGun;
		ArcLEnd [[-569.21,949.78,-14.59],[0.25771,0.331643,-0.885747,-0.197614],[1,-2,2,0],[9E+09,9E+09,9E+09,9E+09,9E+09,9E+09]], v40, seam13, weld13\Weave:=weave1, fine, tWeldGun;
		MoveL [[-569.21,949.78,-8.79],[0.257712,0.331634,-0.88575,-0.197614],[1,-2,2,0],[9E+09,9E+09,9E+09,9E+09,9E+09,9E+09]], vmax, z1, tWeldGun;
		MoveL [[-569.11,978.39,-8.78],[0.257713,0.331647,-0.885744,-0.197616],[1,-2,2,0],[9E+09,9E+09,9E+09,9E+09,9E+09,9E+09]], vmax, z1, tWeldGun;
		ArcLStart [[-569.11,978.38,-14.98],[0.257714,0.331662,-0.885739,-0.197612],[1,-2,2,0],[9E+09,9E+09,9E+09,9E+09,9E+09,9E+09]], v30, seam13, weld13\Weave:=weave1, fine, tWeldGun;
		ArcLEnd [[-569.11,1004.99,-14.97],[0.257723,0.331638,-0.885744,-0.197621],[1,-2,2,0],[9E+09,9E+09,9E+09,9E+09,9E+09,9E+09]], v30, seam13, weld13\Weave:=weave1, fine, tWeldGun;
		MoveL [[-569.11,1004.98,-9.57],[0.257725,0.331632,-0.885746,-0.197618],[1,-2,2,0],[9E+09,9E+09,9E+09,9E+09,9E+09,9E+09]], vmax, z1, tWeldGun;
		MoveL [[-568.66,1030.78,-9.56],[0.257723,0.331657,-0.885737,-0.197616],[1,-2,2,0],[9E+09,9E+09,9E+09,9E+09,9E+09,9E+09]], vmax, z1, tWeldGun;
		ArcLStart [[-569.26,1030.55,-15.38],[0.257732,0.331656,-0.885738,-0.197603],[1,-2,2,0],[9E+09,9E+09,9E+09,9E+09,9E+09,9E+09]], v30, seam13, weld13\Weave:=weave1, fine, tWeldGun;
		ArcLEnd [[-568.86,1056.55,-15.38],[0.257739,0.331642,-0.885741,-0.197603],[1,-2,2,0],[9E+09,9E+09,9E+09,9E+09,9E+09,9E+09]], v30, seam13, weld13\Weave:=weave1, fine, tWeldGun;
		MoveL [[-568.86,1056.55,-6.38],[0.257746,0.331635,-0.885742,-0.197603],[1,-2,2,0],[9E+09,9E+09,9E+09,9E+09,9E+09,9E+09]], vmax, z1, tWeldGun;
		MoveL [[-567.90,1082.34,-6.38],[0.257746,0.331649,-0.885737,-0.197601],[1,-2,2,0],[9E+09,9E+09,9E+09,9E+09,9E+09,9E+09]], vmax, z1, tWeldGun;
		ArcLStart [[-568.70,1082.12,-15.98],[0.257751,0.33165,-0.885737,-0.197592],[1,-2,2,0],[9E+09,9E+09,9E+09,9E+09,9E+09,9E+09]], v20, seam13, weld13\Weave:=weave1, fine, tWeldGun;
		ArcLEnd [[-568.24,1107.52,-15.98],[0.257752,0.331667,-0.885731,-0.19759],[1,-2,2,0],[9E+09,9E+09,9E+09,9E+09,9E+09,9E+09]], v20, seam13, weld13\Weave:=weave1, fine, tWeldGun;
		MoveL [[-568.24,1107.51,-8.98],[0.257762,0.331649,-0.885734,-0.197593],[1,-2,2,0],[9E+09,9E+09,9E+09,9E+09,9E+09,9E+09]], vmax, z1, tWeldGun;
		MoveL [[-568.24,1133.52,-8.97],[0.257758,0.331653,-0.885733,-0.197595],[1,-2,2,0],[9E+09,9E+09,9E+09,9E+09,9E+09,9E+09]], vmax, z1, tWeldGun;
		ArcLStart [[-568.25,1133.51,-15.58],[0.257762,0.331659,-0.885732,-0.197589],[1,-2,2,0],[9E+09,9E+09,9E+09,9E+09,9E+09,9E+09]], v20, seam13, weld13\Weave:=weave1, fine, tWeldGun;
		ArcLEnd [[-568.25,1158.71,-15.60],[0.257768,0.331651,-0.885734,-0.197582],[1,-2,2,0],[9E+09,9E+09,9E+09,9E+09,9E+09,9E+09]], v20, seam13, weld13\Weave:=weave1, fine, tWeldGun;
		MoveL [[-568.24,1158.69,-5.60],[0.257781,0.331624,-0.885741,-0.197583],[1,-2,2,0],[9E+09,9E+09,9E+09,9E+09,9E+09,9E+09]], vmax, z1, tWeldGun;
		MoveL [[-567.89,1183.28,-5.61],[0.257781,0.331645,-0.885735,-0.197572],[1,-2,2,0],[9E+09,9E+09,9E+09,9E+09,9E+09,9E+09]], vmax, z1, tWeldGun;
		ArcLStart [[-568.69,1183.27,-16.02],[0.257789,0.331641,-0.885736,-0.197564],[1,-2,2,0],[9E+09,9E+09,9E+09,9E+09,9E+09,9E+09]], v10, seam13, weld13\Weave:=weave1, fine, tWeldGun;
		ArcLEnd [[-568.49,1207.45,-16.03],[0.257793,0.331641,-0.885736,-0.197559],[1,-2,2,0],[9E+09,9E+09,9E+09,9E+09,9E+09,9E+09]], v10, seam13, weld13\Weave:=weave1, fine, tWeldGun;
		MoveL [[-568.49,1207.45,-8.63],[0.257801,0.331631,-0.885737,-0.197558],[1,-2,2,0],[9E+09,9E+09,9E+09,9E+09,9E+09,9E+09]], vmax, z1, tWeldGun;
		MoveL [[-568.50,1234.87,-8.62],[0.257795,0.331647,-0.885732,-0.197564],[1,-2,2,0],[9E+09,9E+09,9E+09,9E+09,9E+09,9E+09]], vmax, z1, tWeldGun;
		ArcLStart [[-568.49,1234.85,-16.22],[0.25779,0.331666,-0.885728,-0.197556],[1,-2,2,0],[9E+09,9E+09,9E+09,9E+09,9E+09,9E+09]], v10, seam13, weld13\Weave:=weave1, fine, tWeldGun;
		ArcLEnd [[-568.03,1261.25,-16.22],[0.257799,0.331652,-0.88573,-0.19756],[1,-2,2,0],[9E+09,9E+09,9E+09,9E+09,9E+09,9E+09]], v10, seam13, weld13\Weave:=weave1, fine, tWeldGun;
		MoveL [[-568.04,1261.25,-8.21],[0.257811,0.331635,-0.885732,-0.197564],[1,-2,2,0],[9E+09,9E+09,9E+09,9E+09,9E+09,9E+09]], vmax, z1, tWeldGun;
		MoveL [[-567.52,1287.24,-8.21],[0.257803,0.331653,-0.885727,-0.197564],[1,-2,2,0],[9E+09,9E+09,9E+09,9E+09,9E+09,9E+09]], vmax, z1, tWeldGun;
		ArcLStart [[-568.52,1287.23,-15.81],[0.257806,0.331656,-0.885726,-0.197561],[1,-2,2,0],[9E+09,9E+09,9E+09,9E+09,9E+09,9E+09]], v60, seam13, weld13\Weave:=weave1, fine, tWeldGun;
		ArcLEnd [[-568.38,1312.23,-16.00],[0.257804,0.331674,-0.88572,-0.197561],[1,-2,2,0],[9E+09,9E+09,9E+09,9E+09,9E+09,9E+09]], v60, seam13, weld13\Weave:=weave1, fine, tWeldGun;
		MoveL [[-568.37,1312.22,-9.20],[0.257819,0.33164,-0.885728,-0.197564],[1,-2,2,0],[9E+09,9E+09,9E+09,9E+09,9E+09,9E+09]], vmax, z1, tWeldGun;
		MoveL [[-566.34,1338.40,-9.21],[0.257813,0.331671,-0.885721,-0.19755],[1,-2,2,0],[9E+09,9E+09,9E+09,9E+09,9E+09,9E+09]], vmax, z1, tWeldGun;
		ArcLStart [[-567.35,1338.00,-18.39],[0.257823,0.331668,-0.885717,-0.197557],[1,-2,2,0],[9E+09,9E+09,9E+09,9E+09,9E+09,9E+09]], v60, seam13, weld13\Weave:=weave1, fine, tWeldGun;
		ArcLEnd [[-566.97,1362.99,-18.40],[0.257825,0.331676,-0.885715,-0.197551],[1,-2,2,0],[9E+09,9E+09,9E+09,9E+09,9E+09,9E+09]], v60, seam13, weld13\Weave:=weave1, fine, tWeldGun;
		!WorldAccLim\Off;
		MoveL [[-566.97,1362.98,-3.40],[0.257832,0.33166,-0.885719,-0.197554],[1,-2,2,0],[9E+09,9E+09,9E+09,9E+09,9E+09,9E+09]], vmax, z1, tWeldGun;
		MoveJ [[-569.01,1526.90,-0.76],[0.343671,0.343727,-0.853199,-0.189191],[1,-2,2,0],[9E+09,9E+09,9E+09,9E+09,9E+09,9E+09]], vmax, z1, tWeldGun;
		ArcLStart [[-570.01,1526.88,-19.38],[0.343676,0.343732,-0.853197,-0.189182],[1,-2,2,0],[9E+09,9E+09,9E+09,9E+09,9E+09,9E+09]], v30, seam13, weld13\Weave:=weave1, fine, tWeldGun;
		ArcLEnd [[-569.62,1552.28,-19.38],[0.343683,0.343722,-0.853198,-0.189184],[1,-2,2,0],[9E+09,9E+09,9E+09,9E+09,9E+09,9E+09]], v30, seam13, weld13\Weave:=weave1, fine, tWeldGun;
		MoveL [[-569.62,1552.28,-11.37],[0.343694,0.343705,-0.853199,-0.189192],[1,-2,2,0],[9E+09,9E+09,9E+09,9E+09,9E+09,9E+09]], vmax, z1, tWeldGun;
		MoveL [[-569.12,1581.67,-11.38],[0.343681,0.343726,-0.853198,-0.189184],[1,-2,1,0],[9E+09,9E+09,9E+09,9E+09,9E+09,9E+09]], vmax, z1, tWeldGun;
		ArcLStart [[-569.12,1581.67,-19.57],[0.343687,0.343722,-0.853196,-0.189187],[1,-2,2,0],[9E+09,9E+09,9E+09,9E+09,9E+09,9E+09]], v30, seam13, weld13\Weave:=weave1, fine, tWeldGun;
		ArcLEnd [[-568.85,1605.87,-19.56],[0.343691,0.34372,-0.853194,-0.189191],[1,-2,1,0],[9E+09,9E+09,9E+09,9E+09,9E+09,9E+09]], v30, seam13, weld13\Weave:=weave1, fine, tWeldGun;
		MoveL [[-568.85,1605.87,-2.98],[0.343682,0.343726,-0.853196,-0.189187],[1,-1,1,0],[9E+09,9E+09,9E+09,9E+09,9E+09,9E+09]], vmax, z1, tWeldGun;
		MoveL [[-568.53,1630.66,-3.00],[0.343686,0.34372,-0.853198,-0.189182],[1,1,-1,1],[9E+09,9E+09,9E+09,9E+09,9E+09,9E+09]], vmax, z1, tWeldGun;
		ArcLStart [[-570.74,1630.45,-19.81],[0.343708,0.343698,-0.853198,-0.189185],[1,1,-1,1],[9E+09,9E+09,9E+09,9E+09,9E+09,9E+09]], v30, seam13, weld13\Weave:=weave1, fine, tWeldGun;
		ArcLEnd [[-571.08,1657.04,-19.81],[0.343713,0.343698,-0.853195,-0.189186],[1,1,-1,1],[9E+09,9E+09,9E+09,9E+09,9E+09,9E+09]], v30, seam13, weld13\Weave:=weave1, fine, tWeldGun;
		MoveL [[-571.08,1657.05,-10.39],[0.343723,0.343675,-0.853198,-0.189199],[1,1,-1,1],[9E+09,9E+09,9E+09,9E+09,9E+09,9E+09]], vmax, z1, tWeldGun;
		MoveL [[-569.60,1683.62,-10.40],[0.343722,0.343687,-0.853195,-0.189194],[1,1,-1,1],[9E+09,9E+09,9E+09,9E+09,9E+09,9E+09]], vmax, z1, tWeldGun;
		ArcLStart [[-570.40,1683.62,-19.59],[0.343729,0.343674,-0.853196,-0.1892],[1,1,-1,1],[9E+09,9E+09,9E+09,9E+09,9E+09,9E+09]], v30, seam13, weld13\Weave:=weave1, fine, tWeldGun;
		ArcLEnd [[-569.44,1706.01,-19.59],[0.343736,0.343668,-0.853195,-0.1892],[1,1,-1,1],[9E+09,9E+09,9E+09,9E+09,9E+09,9E+09]], v30, seam13, weld13\Weave:=weave1, fine, tWeldGun;
		MoveL [[-569.44,1706.01,-12.58],[0.343736,0.343663,-0.853196,-0.189202],[1,1,-1,1],[9E+09,9E+09,9E+09,9E+09,9E+09,9E+09]], vmax, z1, tWeldGun;
		MoveL [[-568.95,1728.80,-12.59],[0.343738,0.343665,-0.853195,-0.189201],[1,1,-1,1],[9E+09,9E+09,9E+09,9E+09,9E+09,9E+09]], vmax, z1, tWeldGun;
		ArcLStart [[-568.57,1727.28,-19.96],[0.343763,0.34365,-0.853188,-0.189216],[1,1,-1,1],[9E+09,9E+09,9E+09,9E+09,9E+09,9E+09]], v30, seam13, weld13\Weave:=weave1, fine, tWeldGun;
		ArcLEnd [[-568.38,1754.27,-19.94],[0.343779,0.343637,-0.853184,-0.189226],[1,1,-1,1],[9E+09,9E+09,9E+09,9E+09,9E+09,9E+09]], v30, seam13, weld13\Weave:=weave1, fine, tWeldGun;
		MoveL [[-568.37,1754.26,-12.54],[0.343778,0.343636,-0.853186,-0.189221],[1,1,-1,1],[9E+09,9E+09,9E+09,9E+09,9E+09,9E+09]], vmax, z1, tWeldGun;
		MoveL [[-568.19,1780.66,-12.54],[0.343782,0.343632,-0.853186,-0.189224],[1,1,-1,1],[9E+09,9E+09,9E+09,9E+09,9E+09,9E+09]], vmax, z1, tWeldGun;
		ArcLStart [[-568.19,1779.25,-19.93],[0.343783,0.343638,-0.853184,-0.18922],[1,1,-1,1],[9E+09,9E+09,9E+09,9E+09,9E+09,9E+09]], v30, seam13, weld13\Weave:=weave1, fine, tWeldGun;
		ArcLEnd [[-567.11,1804.25,-19.92],[0.343792,0.343628,-0.853182,-0.189228],[1,1,-2,1],[9E+09,9E+09,9E+09,9E+09,9E+09,9E+09]], v30, seam13, weld13\Weave:=weave1, fine, tWeldGun;
		MoveL [[-567.12,1804.23,78.28],[0.343797,0.343622,-0.853184,-0.189223],[1,1,-2,1],[9E+09,9E+09,9E+09,9E+09,9E+09,9E+09]], vmax, z1, tWeldGun;
		ArcLStart [[-567.96,1824.13,-22.58],[0.321693,0.391445,-0.845647,-0.167826],[1,-1,0,0],[9E+09,9E+09,9E+09,9E+09,9E+09,9E+09]], v30, seam13, weld13\Weave:=weave1, fine, tWeldGun;
		ArcLEnd [[-567.85,1853.11,-22.61],[0.321723,0.391404,-0.845654,-0.16783],[1,-1,0,0],[9E+09,9E+09,9E+09,9E+09,9E+09,9E+09]], v30, seam13, weld13\Weave:=weave1, fine, tWeldGun;
		MoveL [[-567.86,1853.06,64.86],[0.321729,0.391441,-0.845624,-0.167883],[1,-1,0,0],[9E+09,9E+09,9E+09,9E+09,9E+09,9E+09]], v30, z1, tWeldGun;
		MoveL [[-589.56,1806.04,41.58],[0.316409,0.386415,-0.856917,-0.127529],[1,-1,0,0],[9E+09,9E+09,9E+09,9E+09,9E+09,9E+09]], v30, z1, tWeldGun;
		MoveL [[-565.44,1418.25,0.00],[0.316355,0.386506,-0.856899,-0.127503],[1,-1,1,0],[9E+09,9E+09,9E+09,9E+09,9E+09,9E+09]], v30, z1, tWeldGun;
		ArcLStart [[-566.84,1418.23,-21.63],[0.31636,0.386522,-0.856891,-0.127501],[1,-1,1,0],[9E+09,9E+09,9E+09,9E+09,9E+09,9E+09]], v30, seam13, weld13\Weave:=weave1, fine, tWeldGun;
		ArcLEnd [[-566.32,1443.02,-21.63],[0.316365,0.386514,-0.856892,-0.127502],[1,-1,1,0],[9E+09,9E+09,9E+09,9E+09,9E+09,9E+09]], v30, seam13, weld13\Weave:=weave1, fine, tWeldGun;
		MoveL [[-566.32,1443.03,10.49],[0.316366,0.386508,-0.856894,-0.127504],[1,-1,1,0],[9E+09,9E+09,9E+09,9E+09,9E+09,9E+09]], v30, z1, tWeldGun;
		MoveL [[-565.57,1462.70,10.49],[0.316366,0.386516,-0.85689,-0.127504],[1,-1,1,0],[9E+09,9E+09,9E+09,9E+09,9E+09,9E+09]], v30, z1, tWeldGun;
		ArcLStart [[-565.57,1456.12,-20.37],[0.316374,0.386523,-0.856885,-0.127501],[1,-1,1,0],[9E+09,9E+09,9E+09,9E+09,9E+09,9E+09]], v30, seam13, weld13\Weave:=weave1, fine, tWeldGun;
		ArcLEnd [[-565.36,1487.97,-20.36],[0.316378,0.386527,-0.856881,-0.127502],[1,-1,1,0],[9E+09,9E+09,9E+09,9E+09,9E+09,9E+09]], v30, seam13, weld13\Weave:=weave1, fine, tWeldGun;
		MoveL [[-565.36,1487.97,2.46],[0.31638,0.386514,-0.856886,-0.127504],[1,-1,1,0],[9E+09,9E+09,9E+09,9E+09,9E+09,9E+09]], v30, z1, tWeldGun;
		MoveL [[-559.76,1655.50,2.46],[0.316384,0.386516,-0.856884,-0.127503],[1,-1,0,0],[9E+09,9E+09,9E+09,9E+09,9E+09,9E+09]], vmax, z1, tWeldGun;
		ArcLStart [[-565.96,1655.48,-22.55],[0.316397,0.386513,-0.856881,-0.127497],[1,-1,1,0],[9E+09,9E+09,9E+09,9E+09,9E+09,9E+09]], v30, seam13, weld13\Weave:=weave1, fine, tWeldGun;
		ArcLEnd [[-566.37,1676.08,-22.53],[0.316408,0.386509,-0.856879,-0.127501],[1,-1,0,0],[9E+09,9E+09,9E+09,9E+09,9E+09,9E+09]], v30, seam13, weld13\Weave:=weave1, fine, tWeldGun;
		MoveL [[-566.36,1676.08,-13.72],[0.316407,0.386508,-0.85688,-0.1275],[1,-1,0,0],[9E+09,9E+09,9E+09,9E+09,9E+09,9E+09]], vmax, z1, tWeldGun;
		MoveL [[-565.20,1705.25,-13.73],[0.316413,0.386506,-0.856879,-0.127497],[1,-1,0,0],[9E+09,9E+09,9E+09,9E+09,9E+09,9E+09]], vmax, z1, tWeldGun;
		ArcLStart [[-565.20,1705.25,-23.32],[0.316413,0.386514,-0.856875,-0.1275],[1,-1,0,0],[9E+09,9E+09,9E+09,9E+09,9E+09,9E+09]], v30, seam13, weld13\Weave:=weave1, fine, tWeldGun;
		ArcLEnd [[-564.28,1720.82,-23.32],[0.316416,0.386511,-0.856874,-0.127501],[1,-1,0,0],[9E+09,9E+09,9E+09,9E+09,9E+09,9E+09]], v30, seam13, weld13\Weave:=weave1, fine, tWeldGun;
		MoveL [[-564.28,1720.81,-13.32],[0.316421,0.3865,-0.856878,-0.1275],[1,-1,0,0],[9E+09,9E+09,9E+09,9E+09,9E+09,9E+09]], vmax, z1, tWeldGun;
		MoveL [[-562.15,1754.27,-13.31],[0.316419,0.386514,-0.856873,-0.127498],[1,-1,0,0],[9E+09,9E+09,9E+09,9E+09,9E+09,9E+09]], vmax, z1, tWeldGun;
		ArcLStart [[-564.55,1753.27,-22.70],[0.316421,0.386527,-0.856865,-0.127503],[1,-1,0,0],[9E+09,9E+09,9E+09,9E+09,9E+09,9E+09]], v30, seam13, weld13\Weave:=weave1, fine, tWeldGun;
		ArcLEnd [[-564.27,1773.06,-22.70],[0.316431,0.386515,-0.856867,-0.127504],[1,-1,0,0],[9E+09,9E+09,9E+09,9E+09,9E+09,9E+09]], v30, seam13, weld13\Weave:=weave1, fine, tWeldGun;
		MoveL [[-564.27,1773.06,-14.70],[0.316433,0.38651,-0.856868,-0.127506],[1,-1,0,0],[9E+09,9E+09,9E+09,9E+09,9E+09,9E+09]], vmax, z1, tWeldGun;
		MoveL [[-562.44,1801.51,-11.84],[0.301948,0.358368,-0.858842,-0.20686],[1,-1,1,0],[9E+09,9E+09,9E+09,9E+09,9E+09,9E+09]], vmax, z1, tWeldGun;
		ArcLStart [[-562.45,1801.50,-21.64],[0.301956,0.358366,-0.858839,-0.206864],[1,-1,1,0],[9E+09,9E+09,9E+09,9E+09,9E+09,9E+09]], v30, seam13, weld13\Weave:=weave1, fine, tWeldGun;
		ArcLEnd [[-561.95,1822.85,-21.66],[0.301963,0.358358,-0.858841,-0.206859],[1,-1,1,0],[9E+09,9E+09,9E+09,9E+09,9E+09,9E+09]], v30, seam13, weld13\Weave:=weave1, fine, tWeldGun;
		MoveL [[-562.07,1822.86,13.32],[0.302053,0.358369,-0.858792,-0.20691],[1,-1,1,0],[9E+09,9E+09,9E+09,9E+09,9E+09,9E+09]], vmax, z1, tWeldGun;
	ENDPROC
PROC rRUNSide1A200()





